LIN {X 0,Y 412.158,Z 270.316,A -85,B 0,C 180,E1 -10502.038,E2 -10502.038} C_VEL
LIN {X 0,Y 411.576,Z 278.2,A -85,B 0,C 180,E1 -10505.303,E2 -10505.303} C_VEL
LIN {X 0,Y 411.175,Z 285.935,A -85,B 0,C 180,E1 -10508.441,E2 -10508.441} C_VEL
LIN {X 0,Y 410.796,Z 293.73,A -85,B 0,C 180,E1 -10511.55,E2 -10511.55} C_VEL
LIN {X 0,Y 410.71,Z 295.781,A -85,B 0,C 180,E1 -10512.362,E2 -10512.362} C_VEL
LIN {X 0,Y 413.099,Z 311.021,A -85,B 0,C 180,E1 -10512.959,E2 -10512.959} C_VEL
LIN {X 0,Y 414.896,Z 323.777,A -85,B 0,C 180,E1 -10513.647,E2 -10513.647} C_VEL
LIN {X 0,Y 414.256,Z 335.412,A -85,B 0,C 180,E1 -10514.377,E2 -10514.377} C_VEL
LIN {X 0,Y 413.495,Z 346.072,A -85,B 0,C 180,E1 -10515.231,E2 -10515.231} C_VEL
LIN {X 0,Y 412.718,Z 356.985,A -85,B 0,C 180,E1 -10516.335,E2 -10516.335} C_VEL
LIN {X 0,Y 412.142,Z 365.905,A -85,B 0,C 180,E1 -10517.444,E2 -10517.444} C_VEL
LIN {X 0,Y 411.367,Z 375.608,A -85,B 0,C 180,E1 -10518.92,E2 -10518.92} C_VEL
LIN {X 0,Y 410.824,Z 383.345,A -85,B 0,C 180,E1 -10520.4,E2 -10520.4} C_VEL
LIN {X 0,Y 410.352,Z 390.488,A -85,B 0,C 180,E1 -10522.126,E2 -10522.126} C_VEL
LIN {X 0,Y 410.176,Z 395.252,A -85,B 0,C 180,E1 -10523.607,E2 -10523.607} C_VEL
LIN {X 0,Y 410.095,Z 398.897,A -85,B 0,C 180,E1 -10525.086,E2 -10525.086} C_VEL
LIN {X 0,Y 409.954,Z 400.772,A -85,B 0,C 180,E1 -10526.069,E2 -10526.069} C_VEL
LIN {X 0,Y 410.007,Z 402.189,A -85,B 0,C 180,E1 -10527.054,E2 -10527.054} C_VEL
LIN {X 0,Y 409.988,Z 403.197,A -85,B 0,C 180,E1 -10528.037,E2 -10528.037} C_VEL
LIN {X 0,Y 409.958,Z 403.812,A -85,B 0,C 180,E1 -10529.019,E2 -10529.019} C_VEL
LIN {X 0,Y 409.967,Z 404.032,A -85,B 0,C 180,E1 -10530.001,E2 -10530.001} C_VEL
LIN {X 0,Y 409.959,Z 403.815,A -85,B 0,C 180,E1 -10530.984,E2 -10530.984} C_VEL
LIN {X 0,Y 409.989,Z 403.204,A -85,B 0,C 180,E1 -10531.966,E2 -10531.966} C_VEL
LIN {X 0,Y 410.007,Z 402.201,A -85,B 0,C 180,E1 -10532.949,E2 -10532.949} C_VEL
LIN {X 0,Y 409.955,Z 400.787,A -85,B 0,C 180,E1 -10533.933,E2 -10533.933} C_VEL
LIN {X 0,Y 410.108,Z 397.83,A -85,B 0,C 180,E1 -10535.41,E2 -10535.41} C_VEL
LIN {X 0,Y 410.199,Z 393.819,A -85,B 0,C 180,E1 -10536.89,E2 -10536.89} C_VEL
LIN {X 0,Y 410.552,Z 387.661,A -85,B 0,C 180,E1 -10538.616,E2 -10538.616} C_VEL
LIN {X 0,Y 410.995,Z 380.937,A -85,B 0,C 180,E1 -10540.096,E2 -10540.096} C_VEL
LIN {X 0,Y 411.603,Z 372.598,A -85,B 0,C 180,E1 -10541.575,E2 -10541.575} C_VEL
LIN {X 0,Y 412.222,Z 364.05,A -85,B 0,C 180,E1 -10542.807,E2 -10542.807} C_VEL
LIN {X 0,Y 412.945,Z 354.466,A -85,B 0,C 180,E1 -10543.934,E2 -10543.934} C_VEL
LIN {X 0,Y 413.699,Z 343.045,A -85,B 0,C 180,E1 -10545.016,E2 -10545.016} C_VEL
LIN {X 0,Y 414.479,Z 331.604,A -85,B 0,C 180,E1 -10545.869,E2 -10545.869} C_VEL
LIN {X 0,Y 414.807,Z 323.36,A -85,B 0,C 180,E1 -10546.359,E2 -10546.359} C_VEL
LIN {X 0,Y 412.936,Z 309.911,A -85,B 0,C 180,E1 -10547.061,E2 -10547.061} C_VEL
LIN {X 0,Y 410.806,Z 297.017,A -85,B 0,C 180,E1 -10547.536,E2 -10547.536} C_VEL
LIN {X 0,Y 410.688,Z 295.908,A -85,B 0,C 180,E1 -10547.565,E2 -10547.565} C_VEL
LIN {X 0,Y 411.053,Z 288.417,A -85,B 0,C 180,E1 -10550.519,E2 -10550.519} C_VEL
LIN {X 0,Y 411.401,Z 280.488,A -85,B 0,C 180,E1 -10553.67,E2 -10553.67} C_VEL
LIN {X 0,Y 411.91,Z 272.527,A -85,B 0,C 180,E1 -10556.883,E2 -10556.883} C_VEL
LIN {X 0,Y 412.427,Z 264.541,A -85,B 0,C 180,E1 -10560.18,E2 -10560.18} C_VEL
LIN {X 0,Y 412.928,Z 257.914,A -85,B 0,C 180,E1 -10563.001,E2 -10563.001} C_VEL
LIN {X 0,Y 413.391,Z 251.345,A -85,B 0,C 180,E1 -10565.913,E2 -10565.913} C_VEL
LIN {X 0,Y 413.002,Z 247.385,A -85,B 0,C 180,E1 -10567.78,E2 -10567.78} C_VEL
LIN {X 0,Y 411.812,Z 240.314,A -85,B 0,C 180,E1 -10571.331,E2 -10571.331} C_VEL
LIN {X 0,Y 411.213,Z 237.266,A -85,B 0,C 180,E1 -10572.958,E2 -10572.958} C_VEL
LIN {X 0,Y 411.175,Z 237.273,A -85,B 0,C 180,E1 -10575.882,E2 -10575.882} C_VEL
LIN {X 0,Y 411.17,Z 237.27,A -85,B 0,C 180,E1 -10578.772,E2 -10578.772} C_VEL
LIN {X 0,Y 411.198,Z 237.263,A -85,B 0,C 180,E1 -10582.027,E2 -10582.027} C_VEL
LIN {X 0,Y 411.199,Z 237.261,A -85,B 0,C 180,E1 -10585.666,E2 -10585.666} C_VEL
LIN {X 0,Y 411.194,Z 237.263,A -85,B 0,C 180,E1 -10589.153,E2 -10589.153} C_VEL
LIN {X 0,Y 411.215,Z 237.263,A -85,B 0,C 180,E1 -10592.519,E2 -10592.519} C_VEL
LIN {X 0,Y 411.225,Z 237.262,A -85,B 0,C 180,E1 -10595.785,E2 -10595.785} C_VEL
LIN {X 0,Y 411.204,Z 237.262,A -85,B 0,C 180,E1 -10598.966,E2 -10598.966} C_VEL
LIN {X 0,Y 411.237,Z 237.262,A -85,B 0,C 180,E1 -10602.084,E2 -10602.084} C_VEL
LIN {X 0,Y 411.236,Z 237.257,A -85,B 0,C 180,E1 -10605.147,E2 -10605.147} C_VEL
LIN {X 0,Y 411.28,Z 237.254,A -85,B 0,C 180,E1 -10608.167,E2 -10608.167} C_VEL
LIN {X 0,Y 411.446,Z 237.234,A -85,B 0,C 180,E1 -10612.192,E2 -10612.192} C_VEL
LIN {X 0,Y 411.473,Z 237.231,A -85,B 0,C 180,E1 -10614.118,E2 -10614.118} C_VEL
LIN {X 0,Y 411.518,Z 237.225,A -85,B 0,C 180,E1 -10618.043,E2 -10618.043} C_VEL
LIN {X 0,Y 411.644,Z 237.209,A -85,B 0,C 180,E1 -10620,E2 -10620} C_VEL
LIN {X 0,Y 411.452,Z 237.232,A -85,B 0,C 180,E1 -10622.937,E2 -10622.937} C_VEL
LIN {X 0,Y 411.393,Z 237.239,A -85,B 0,C 180,E1 -10626.868,E2 -10626.868} C_VEL
LIN {X 0,Y 411.292,Z 237.252,A -85,B 0,C 180,E1 -10629.839,E2 -10629.839} C_VEL
LIN {X 0,Y 411.314,Z 237.252,A -85,B 0,C 180,E1 -10633.104,E2 -10633.104} C_VEL
LIN {X 0,Y 411.266,Z 237.257,A -85,B 0,C 180,E1 -10636.889,E2 -10636.889} C_VEL
LIN {X 0,Y 411.239,Z 237.258,A -85,B 0,C 180,E1 -10639.987,E2 -10639.987} C_VEL
LIN {X 0,Y 411.194,Z 237.266,A -85,B 0,C 180,E1 -10643.148,E2 -10643.148} C_VEL
LIN {X 0,Y 411.171,Z 237.267,A -85,B 0,C 180,E1 -10646.386,E2 -10646.386} C_VEL
LIN {X 0,Y 411.204,Z 237.261,A -85,B 0,C 180,E1 -10649.713,E2 -10649.713} C_VEL
LIN {X 0,Y 411.214,Z 237.262,A -85,B 0,C 180,E1 -10653.155,E2 -10653.155} C_VEL
LIN {X 0,Y 411.199,Z 237.266,A -85,B 0,C 180,E1 -10656.552,E2 -10656.552} C_VEL
LIN {X 0,Y 411.214,Z 237.262,A -85,B 0,C 180,E1 -10659.726,E2 -10659.726} C_VEL
LIN {X 0,Y 411.178,Z 237.265,A -85,B 0,C 180,E1 -10663.133,E2 -10663.133} C_VEL
LIN {X 0,Y 411.17,Z 237.268,A -85,B 0,C 180,E1 -10665.881,E2 -10665.881} C_VEL
LIN {X 0,Y 411.164,Z 237.267,A -85,B 0,C 180,E1 -10669.492,E2 -10669.492} C_VEL
LIN {X 0,Y 411.192,Z 237.267,A -85,B 0,C 180,E1 -10672.024,E2 -10672.024} C_VEL
LIN {X 0,Y 411.21,Z 237.262,A -85,B 0,C 180,E1 -10675.122,E2 -10675.122} C_VEL
LIN {X 0,Y 411.107,Z 237.277,A -85,B 0,C 180,E1 -10677.996,E2 -10677.996} C_VEL
LIN {X 0,Y 410.789,Z 237.318,A -85,B 0,C 180,E1 -10681.376,E2 -10681.376} C_VEL
LIN {X 0,Y 410.632,Z 237.497,A -85,B 0,C 180,E1 -10682.872,E2 -10682.872} C_VEL
LIN {X 0,Y 410.568,Z 240.288,A -85,B 0,C 180,E1 -10685.742,E2 -10685.742} C_VEL
LIN {X 0,Y 410.475,Z 243.402,A -85,B 0,C 180,E1 -10688.926,E2 -10688.926} C_VEL
LIN {X 0,Y 410.409,Z 246.589,A -85,B 0,C 180,E1 -10692.045,E2 -10692.045} C_VEL
LIN {X 0,Y 410.381,Z 249.825,A -85,B 0,C 180,E1 -10695.113,E2 -10695.113} C_VEL
LIN {X 0,Y 410.411,Z 251.602,A -85,B 0,C 180,E1 -10696.745,E2 -10696.745} C_VEL
LIN {X 0,Y 413.741,Z 265.221,A -85,B 0,C 180,E1 -10697.347,E2 -10697.347} C_VEL
LIN {X 0,Y 415.318,Z 272.966,A -85,B 0,C 180,E1 -10697.776,E2 -10697.776} C_VEL
LIN {X 0,Y 414.783,Z 285.252,A -85,B 0,C 180,E1 -10698.515,E2 -10698.515} C_VEL
LIN {X 0,Y 414.047,Z 297.573,A -85,B 0,C 180,E1 -10699.485,E2 -10699.485} C_VEL
LIN {X 0,Y 413.416,Z 307.511,A -85,B 0,C 180,E1 -10700.482,E2 -10700.482} C_VEL
LIN {X 0,Y 412.804,Z 317.143,A -85,B 0,C 180,E1 -10701.678,E2 -10701.678} C_VEL
LIN {X 0,Y 412.051,Z 326.69,A -85,B 0,C 180,E1 -10703.142,E2 -10703.142} C_VEL
LIN {X 0,Y 411.438,Z 334.306,A -85,B 0,C 180,E1 -10704.608,E2 -10704.608} C_VEL
LIN {X 0,Y 410.884,Z 340.421,A -85,B 0,C 180,E1 -10706.075,E2 -10706.075} C_VEL
LIN {X 0,Y 410.502,Z 345.28,A -85,B 0,C 180,E1 -10707.545,E2 -10707.545} C_VEL
LIN {X 0,Y 410.231,Z 349.036,A -85,B 0,C 180,E1 -10709.017,E2 -10709.017} C_VEL
LIN {X 0,Y 410.163,Z 350.969,A -85,B 0,C 180,E1 -10709.999,E2 -10709.999} C_VEL
LIN {X 0,Y 410.148,Z 352.495,A -85,B 0,C 180,E1 -10710.98,E2 -10710.98} C_VEL
LIN {X 0,Y 410.143,Z 353.592,A -85,B 0,C 180,E1 -10711.963,E2 -10711.963} C_VEL
LIN {X 0,Y 410.195,Z 354.28,A -85,B 0,C 180,E1 -10712.945,E2 -10712.945} C_VEL
LIN {X 0,Y 410.11,Z 354.543,A -85,B 0,C 180,E1 -10714.914,E2 -10714.914} C_VEL
LIN {X 0,Y 410.212,Z 353.644,A -85,B 0,C 180,E1 -10716.435,E2 -10716.435} C_VEL
LIN {X 0,Y 410.296,Z 351.92,A -85,B 0,C 180,E1 -10717.875,E2 -10717.875} C_VEL
LIN {X 0,Y 410.485,Z 348.979,A -85,B 0,C 180,E1 -10719.466,E2 -10719.466} C_VEL
LIN {X 0,Y 409.963,Z 347.209,A -85,B 0,C 180,E1 -10720.249,E2 -10720.249} C_VEL
LIN {X 0,Y 407.393,Z 343.929,A -85,B 0,C 180,E1 -10721.513,E2 -10721.513} C_VEL
LIN {X 0,Y 404.911,Z 340.075,A -85,B 0,C 180,E1 -10722.754,E2 -10722.754} C_VEL
LIN {X 0,Y 404.534,Z 337.241,A -85,B 0,C 180,E1 -10723.49,E2 -10723.49} C_VEL
LIN {X 0,Y 405.238,Z 329.743,A -85,B 0,C 180,E1 -10725.077,E2 -10725.077} C_VEL
LIN {X 0,Y 406.067,Z 320.767,A -85,B 0,C 180,E1 -10726.592,E2 -10726.592} C_VEL
LIN {X 0,Y 406.922,Z 311.461,A -85,B 0,C 180,E1 -10727.851,E2 -10727.851} C_VEL
LIN {X 0,Y 407.693,Z 301.065,A -85,B 0,C 180,E1 -10728.987,E2 -10728.987} C_VEL
LIN {X 0,Y 408.603,Z 289.481,A -85,B 0,C 180,E1 -10729.988,E2 -10729.988} C_VEL
LIN {X 0,Y 409.132,Z 277.866,A -85,B 0,C 180,E1 -10730.774,E2 -10730.774} C_VEL
LIN {X 0,Y 409.283,Z 275.137,A -85,B 0,C 180,E1 -10730.924,E2 -10730.924} C_VEL
LIN {X 0,Y 406.594,Z 263.548,A -85,B 0,C 180,E1 -10731.625,E2 -10731.625} C_VEL
LIN {X 0,Y 403.358,Z 252.181,A -85,B 0,C 180,E1 -10732.198,E2 -10732.198} C_VEL
LIN {X 0,Y 403.446,Z 248.467,A -85,B 0,C 180,E1 -10735.815,E2 -10735.815} C_VEL
LIN {X 0,Y 403.577,Z 244.876,A -85,B 0,C 180,E1 -10739.458,E2 -10739.458} C_VEL
LIN {X 0,Y 403.601,Z 241.861,A -85,B 0,C 180,E1 -10742.669,E2 -10742.669} C_VEL
LIN {X 0,Y 403.723,Z 239.598,A -85,B 0,C 180,E1 -10745.097,E2 -10745.097} C_VEL
LIN {X 0,Y 403.816,Z 238.188,A -85,B 0,C 180,E1 -10746.814,E2 -10746.814} C_VEL
LIN {X 0,Y 404.085,Z 238.149,A -85,B 0,C 180,E1 -10750.069,E2 -10750.069} C_VEL
LIN {X 0,Y 404.145,Z 238.144,A -85,B 0,C 180,E1 -10753.082,E2 -10753.082} C_VEL
LIN {X 0,Y 404.14,Z 238.146,A -85,B 0,C 180,E1 -10755.925,E2 -10755.925} C_VEL
LIN {X 0,Y 404.107,Z 238.148,A -85,B 0,C 180,E1 -10758.633,E2 -10758.633} C_VEL
LIN {X 0,Y 404.145,Z 238.142,A -85,B 0,C 180,E1 -10761.491,E2 -10761.491} C_VEL
LIN {X 0,Y 404.177,Z 238.138,A -85,B 0,C 180,E1 -10764.983,E2 -10764.983} C_VEL
LIN {X 0,Y 404.132,Z 238.143,A -85,B 0,C 180,E1 -10768.553,E2 -10768.553} C_VEL
LIN {X 0,Y 404.186,Z 238.137,A -85,B 0,C 180,E1 -10771.999,E2 -10771.999} C_VEL
LIN {X 0,Y 404.167,Z 238.14,A -85,B 0,C 180,E1 -10775.333,E2 -10775.333} C_VEL
LIN {X 0,Y 404.128,Z 238.145,A -85,B 0,C 180,E1 -10778.58,E2 -10778.58} C_VEL
LIN {X 0,Y 404.199,Z 238.135,A -85,B 0,C 180,E1 -10781.761,E2 -10781.761} C_VEL
LIN {X 0,Y 404.195,Z 238.136,A -85,B 0,C 180,E1 -10784.881,E2 -10784.881} C_VEL
LIN {X 0,Y 404.244,Z 238.129,A -85,B 0,C 180,E1 -10787.958,E2 -10787.958} C_VEL
LIN {X 0,Y 404.422,Z 238.111,A -85,B 0,C 180,E1 -10792.099,E2 -10792.099} C_VEL
LIN {X 0,Y 404.429,Z 238.111,A -85,B 0,C 180,E1 -10794.015,E2 -10794.015} C_VEL
LIN {X 0,Y 404.472,Z 238.101,A -85,B 0,C 180,E1 -10798.008,E2 -10798.008} C_VEL
LIN {X 0,Y 404.596,Z 238.087,A -85,B 0,C 180,E1 -10800,E2 -10800} C_VEL
LIN {X 0,Y 404.413,Z 238.109,A -85,B 0,C 180,E1 -10802.988,E2 -10802.988} C_VEL
LIN {X 0,Y 404.428,Z 238.107,A -85,B 0,C 180,E1 -10805.985,E2 -10805.985} C_VEL
LIN {X 0,Y 404.411,Z 238.109,A -85,B 0,C 180,E1 -10807.991,E2 -10807.991} C_VEL
LIN {X 0,Y 404.244,Z 238.133,A -85,B 0,C 180,E1 -10812.042,E2 -10812.042} C_VEL
LIN {X 0,Y 404.194,Z 238.136,A -85,B 0,C 180,E1 -10815.118,E2 -10815.118} C_VEL
LIN {X 0,Y 404.199,Z 238.136,A -85,B 0,C 180,E1 -10818.239,E2 -10818.239} C_VEL
LIN {X 0,Y 404.127,Z 238.145,A -85,B 0,C 180,E1 -10821.42,E2 -10821.42} C_VEL
LIN {X 0,Y 404.166,Z 238.14,A -85,B 0,C 180,E1 -10824.666,E2 -10824.666} C_VEL
LIN {X 0,Y 404.188,Z 238.138,A -85,B 0,C 180,E1 -10828,E2 -10828} C_VEL
LIN {X 0,Y 404.136,Z 238.146,A -85,B 0,C 180,E1 -10831.56,E2 -10831.56} C_VEL
LIN {X 0,Y 404.175,Z 238.139,A -85,B 0,C 180,E1 -10835.017,E2 -10835.017} C_VEL
LIN {X 0,Y 404.145,Z 238.144,A -85,B 0,C 180,E1 -10838.758,E2 -10838.758} C_VEL
LIN {X 0,Y 404.11,Z 238.149,A -85,B 0,C 180,E1 -10841.6,E2 -10841.6} C_VEL
LIN {X 0,Y 404.137,Z 238.146,A -85,B 0,C 180,E1 -10844.523,E2 -10844.523} C_VEL
LIN {X 0,Y 404.152,Z 238.286,A -85,B 0,C 180,E1 -10845.839,E2 -10845.839} C_VEL
LIN {X 0,Y 405.143,Z 243.346,A -85,B 0,C 180,E1 -10848.765,E2 -10848.765} C_VEL
LIN {X 0,Y 406.197,Z 249.585,A -85,B 0,C 180,E1 -10852.108,E2 -10852.108} C_VEL
LIN {X 0,Y 406.557,Z 253.389,A -85,B 0,C 180,E1 -10854.005,E2 -10854.005} C_VEL
LIN {X 0,Y 406.046,Z 259.761,A -85,B 0,C 180,E1 -10856.963,E2 -10856.963} C_VEL
LIN {X 0,Y 405.374,Z 266.817,A -85,B 0,C 180,E1 -10860.095,E2 -10860.095} C_VEL
LIN {X 0,Y 404.903,Z 273.956,A -85,B 0,C 180,E1 -10863.175,E2 -10863.175} C_VEL
LIN {X 0,Y 404.259,Z 283.395,A -85,B 0,C 180,E1 -10867.132,E2 -10867.132} C_VEL
LIN {X 0,Y 403.903,Z 290.359,A -85,B 0,C 180,E1 -10869.987,E2 -10869.987} C_VEL
LIN {X 0,Y 403.661,Z 295.493,A -85,B 0,C 180,E1 -10872.05,E2 -10872.05} C_VEL
LIN {X 0,Y 405.902,Z 308.96,A -85,B 0,C 180,E1 -10872.562,E2 -10872.562} C_VEL
LIN {X 0,Y 407.69,Z 321.978,A -85,B 0,C 180,E1 -10873.257,E2 -10873.257} C_VEL
LIN {X 0,Y 408.009,Z 326.19,A -85,B 0,C 180,E1 -10873.515,E2 -10873.515} C_VEL
LIN {X 0,Y 407.144,Z 338.416,A -85,B 0,C 180,E1 -10874.354,E2 -10874.354} C_VEL
LIN {X 0,Y 406.287,Z 350.067,A -85,B 0,C 180,E1 -10875.386,E2 -10875.386} C_VEL
LIN {X 0,Y 405.557,Z 359.842,A -85,B 0,C 180,E1 -10876.472,E2 -10876.472} C_VEL
LIN {X 0,Y 404.878,Z 369.022,A -85,B 0,C 180,E1 -10877.725,E2 -10877.725} C_VEL
LIN {X 0,Y 404.114,Z 377.979,A -85,B 0,C 180,E1 -10879.226,E2 -10879.226} C_VEL
LIN {X 0,Y 403.611,Z 385.201,A -85,B 0,C 180,E1 -10880.733,E2 -10880.733} C_VEL
LIN {X 0,Y 403.299,Z 390.084,A -85,B 0,C 180,E1 -10881.988,E2 -10881.988} C_VEL
LIN {X 0,Y 403.068,Z 395.288,A -85,B 0,C 180,E1 -10883.652,E2 -10883.652} C_VEL
LIN {X 0,Y 403.007,Z 398.478,A -85,B 0,C 180,E1 -10884.999,E2 -10884.999} C_VEL
LIN {X 0,Y 402.877,Z 400.351,A -85,B 0,C 180,E1 -10886,E2 -10886} C_VEL
LIN {X 0,Y 402.908,Z 401.764,A -85,B 0,C 180,E1 -10887.002,E2 -10887.002} C_VEL
LIN {X 0,Y 402.921,Z 402.773,A -85,B 0,C 180,E1 -10888.002,E2 -10888.002} C_VEL
LIN {X 0,Y 402.884,Z 403.387,A -85,B 0,C 180,E1 -10889.002,E2 -10889.002} C_VEL
LIN {X 0,Y 402.89,Z 403.606,A -85,B 0,C 180,E1 -10890.001,E2 -10890.001} C_VEL
LIN {X 0,Y 402.921,Z 402.776,A -85,B 0,C 180,E1 -10892.001,E2 -10892.001} C_VEL
LIN {X 0,Y 402.909,Z 401.769,A -85,B 0,C 180,E1 -10893.001,E2 -10893.001} C_VEL
LIN {X 0,Y 402.877,Z 400.354,A -85,B 0,C 180,E1 -10894.003,E2 -10894.003} C_VEL
LIN {X 0,Y 403.007,Z 397.391,A -85,B 0,C 180,E1 -10895.505,E2 -10895.505} C_VEL
LIN {X 0,Y 403.118,Z 393.373,A -85,B 0,C 180,E1 -10897.011,E2 -10897.011} C_VEL
LIN {X 0,Y 403.518,Z 387.204,A -85,B 0,C 180,E1 -10898.767,E2 -10898.767} C_VEL
LIN {X 0,Y 403.967,Z 380.466,A -85,B 0,C 180,E1 -10900.274,E2 -10900.274} C_VEL
LIN {X 0,Y 404.61,Z 372.111,A -85,B 0,C 180,E1 -10901.778,E2 -10901.778} C_VEL
LIN {X 0,Y 405.238,Z 363.536,A -85,B 0,C 180,E1 -10903.031,E2 -10903.031} C_VEL
LIN {X 0,Y 406.022,Z 353.452,A -85,B 0,C 180,E1 -10904.227,E2 -10904.227} C_VEL
LIN {X 0,Y 406.791,Z 342.474,A -85,B 0,C 180,E1 -10905.277,E2 -10905.277} C_VEL
LIN {X 0,Y 407.637,Z 331.106,A -85,B 0,C 180,E1 -10906.134,E2 -10906.134} C_VEL
LIN {X 0,Y 407.919,Z 324.481,A -85,B 0,C 180,E1 -10906.542,E2 -10906.542} C_VEL
LIN {X 0,Y 406.056,Z 310.699,A -85,B 0,C 180,E1 -10907.292,E2 -10907.292} C_VEL
LIN {X 0,Y 403.915,Z 297.479,A -85,B 0,C 180,E1 -10907.808,E2 -10907.808} C_VEL
LIN {X 0,Y 403.625,Z 295.48,A -85,B 0,C 180,E1 -10907.873,E2 -10907.873} C_VEL
LIN {X 0,Y 404.072,Z 286.681,A -85,B 0,C 180,E1 -10911.425,E2 -10911.425} C_VEL
LIN {X 0,Y 404.628,Z 276.913,A -85,B 0,C 180,E1 -10915.419,E2 -10915.419} C_VEL
LIN {X 0,Y 405.137,Z 269.504,A -85,B 0,C 180,E1 -10918.494,E2 -10918.494} C_VEL
LIN {X 0,Y 405.753,Z 261.477,A -85,B 0,C 180,E1 -10921.927,E2 -10921.927} C_VEL
LIN {X 0,Y 406.26,Z 254.965,A -85,B 0,C 180,E1 -10924.813,E2 -10924.813} C_VEL
LIN {X 0,Y 406.334,Z 251.056,A -85,B 0,C 180,E1 -10926.629,E2 -10926.629} C_VEL
LIN {X 0,Y 405.527,Z 245.689,A -85,B 0,C 180,E1 -10929.29,E2 -10929.29} C_VEL
LIN {X 0,Y 404.417,Z 239.27,A -85,B 0,C 180,E1 -10932.669,E2 -10932.669} C_VEL
LIN {X 0,Y 404.159,Z 238.146,A -85,B 0,C 180,E1 -10933.338,E2 -10933.338} C_VEL
LIN {X 0,Y 404.16,Z 238.143,A -85,B 0,C 180,E1 -10936.917,E2 -10936.917} C_VEL
LIN {X 0,Y 404.176,Z 238.14,A -85,B 0,C 180,E1 -10939.956,E2 -10939.956} C_VEL
LIN {X 0,Y 404.142,Z 238.142,A -85,B 0,C 180,E1 -10943.126,E2 -10943.126} C_VEL
LIN {X 0,Y 404.144,Z 238.143,A -85,B 0,C 180,E1 -10946.188,E2 -10946.188} C_VEL
LIN {X 0,Y 404.15,Z 238.14,A -85,B 0,C 180,E1 -10949.715,E2 -10949.715} C_VEL
LIN {X 0,Y 404.158,Z 238.14,A -85,B 0,C 180,E1 -10953.12,E2 -10953.12} C_VEL
LIN {X 0,Y 404.173,Z 238.141,A -85,B 0,C 180,E1 -10956.426,E2 -10956.426} C_VEL
LIN {X 0,Y 404.199,Z 238.137,A -85,B 0,C 180,E1 -10959.875,E2 -10959.875} C_VEL
LIN {X 0,Y 404.181,Z 238.136,A -85,B 0,C 180,E1 -10963.013,E2 -10963.013} C_VEL
LIN {X 0,Y 404.291,Z 238.122,A -85,B 0,C 180,E1 -10966.939,E2 -10966.939} C_VEL
LIN {X 0,Y 404.252,Z 238.131,A -85,B 0,C 180,E1 -10969.988,E2 -10969.988} C_VEL
LIN {X 0,Y 404.393,Z 238.111,A -85,B 0,C 180,E1 -10973.013,E2 -10973.013} C_VEL
LIN {X 0,Y 404.285,Z 238.124,A -85,B 0,C 180,E1 -10975.014,E2 -10975.014} C_VEL
LIN {X 0,Y 404.487,Z 238.101,A -85,B 0,C 180,E1 -10978.009,E2 -10978.009} C_VEL
LIN {X 0,Y 404.613,Z 238.085,A -85,B 0,C 180,E1 -10980,E2 -10980} C_VEL
LIN {X 0,Y 404.41,Z 238.11,A -85,B 0,C 180,E1 -10982.989,E2 -10982.989} C_VEL
LIN {X 0,Y 404.344,Z 238.118,A -85,B 0,C 180,E1 -10986.989,E2 -10986.989} C_VEL
LIN {X 0,Y 404.258,Z 238.127,A -85,B 0,C 180,E1 -10990.012,E2 -10990.012} C_VEL
LIN {X 0,Y 404.275,Z 238.128,A -85,B 0,C 180,E1 -10993.211,E2 -10993.211} C_VEL
LIN {X 0,Y 404.224,Z 238.135,A -85,B 0,C 180,E1 -10997.007,E2 -10997.007} C_VEL
LIN {X 0,Y 404.172,Z 238.139,A -85,B 0,C 180,E1 -11000.351,E2 -11000.351} C_VEL
LIN {X 0,Y 404.155,Z 238.14,A -85,B 0,C 180,E1 -11003.576,E2 -11003.576} C_VEL
LIN {X 0,Y 404.105,Z 238.149,A -85,B 0,C 180,E1 -11006.884,E2 -11006.884} C_VEL
LIN {X 0,Y 404.151,Z 238.143,A -85,B 0,C 180,E1 -11010.285,E2 -11010.285} C_VEL
LIN {X 0,Y 404.152,Z 238.141,A -85,B 0,C 180,E1 -11013.812,E2 -11013.812} C_VEL
LIN {X 0,Y 404.142,Z 238.144,A -85,B 0,C 180,E1 -11016.874,E2 -11016.874} C_VEL
LIN {X 0,Y 404.155,Z 238.143,A -85,B 0,C 180,E1 -11020.08,E2 -11020.08} C_VEL
LIN {X 0,Y 404.157,Z 238.139,A -85,B 0,C 180,E1 -11023.083,E2 -11023.083} C_VEL
LIN {X 0,Y 404.127,Z 238.146,A -85,B 0,C 180,E1 -11025.921,E2 -11025.921} C_VEL
LIN {X 0,Y 404.107,Z 238.146,A -85,B 0,C 180,E1 -11028.632,E2 -11028.632} C_VEL
LIN {X 0,Y 404.146,Z 238.142,A -85,B 0,C 180,E1 -11031.494,E2 -11031.494} C_VEL
LIN {X 0,Y 404.181,Z 238.137,A -85,B 0,C 180,E1 -11034.982,E2 -11034.982} C_VEL
LIN {X 0,Y 404.106,Z 238.148,A -85,B 0,C 180,E1 -11037.374,E2 -11037.374} C_VEL
LIN {X 0,Y 403.861,Z 238.177,A -85,B 0,C 180,E1 -11040.471,E2 -11040.471} C_VEL
LIN {X 0,Y 403.581,Z 238.217,A -85,B 0,C 180,E1 -11042.639,E2 -11042.639} C_VEL
LIN {X 0,Y 403.551,Z 240.636,A -85,B 0,C 180,E1 -11045.292,E2 -11045.292} C_VEL
LIN {X 0,Y 403.409,Z 243.794,A -85,B 0,C 180,E1 -11048.539,E2 -11048.539} C_VEL
LIN {X 0,Y 403.349,Z 247.016,A -85,B 0,C 180,E1 -11051.72,E2 -11051.72} C_VEL
LIN {X 0,Y 403.368,Z 249.156,A -85,B 0,C 180,E1 -11053.812,E2 -11053.812} C_VEL
LIN {X 0,Y 403.343,Z 252.005,A -85,B 0,C 180,E1 -11056.457,E2 -11056.457} C_VEL
LIN {X 0,Y 406.664,Z 265.573,A -85,B 0,C 180,E1 -11057.069,E2 -11057.069} C_VEL
LIN {X 0,Y 408.436,Z 274.588,A -85,B 0,C 180,E1 -11057.586,E2 -11057.586} C_VEL
LIN {X 0,Y 407.891,Z 286.345,A -85,B 0,C 180,E1 -11058.318,E2 -11058.318} C_VEL
LIN {X 0,Y 407.222,Z 297.129,A -85,B 0,C 180,E1 -11059.181,E2 -11059.181} C_VEL
LIN {X 0,Y 406.486,Z 308.339,A -85,B 0,C 180,E1 -11060.318,E2 -11060.318} C_VEL
LIN {X 0,Y 405.838,Z 317.906,A -85,B 0,C 180,E1 -11061.534,E2 -11061.534} C_VEL
LIN {X 0,Y 405.055,Z 327.394,A -85,B 0,C 180,E1 -11063.022,E2 -11063.022} C_VEL
LIN {X 0,Y 404.413,Z 334.944,A -85,B 0,C 180,E1 -11064.514,E2 -11064.514} C_VEL
LIN {X 0,Y 403.825,Z 341.021,A -85,B 0,C 180,E1 -11066.007,E2 -11066.007} C_VEL
LIN {X 0,Y 403.445,Z 345.842,A -85,B 0,C 180,E1 -11067.503,E2 -11067.503} C_VEL
LIN {X 0,Y 403.175,Z 349.562,A -85,B 0,C 180,E1 -11069,E2 -11069} C_VEL
LIN {X 0,Y 403.106,Z 351.479,A -85,B 0,C 180,E1 -11069.999,E2 -11069.999} C_VEL
LIN {X 0,Y 403.063,Z 352.989,A -85,B 0,C 180,E1 -11070.998,E2 -11070.998} C_VEL
LIN {X 0,Y 403.126,Z 354.729,A -85,B 0,C 180,E1 -11072.997,E2 -11072.997} C_VEL
LIN {X 0,Y 403.045,Z 354.961,A -85,B 0,C 180,E1 -11075,E2 -11075} C_VEL
LIN {X 0,Y 403.143,Z 354.118,A -85,B 0,C 180,E1 -11076.44,E2 -11076.44} C_VEL
LIN {X 0,Y 403.234,Z 352.279,A -85,B 0,C 180,E1 -11078.013,E2 -11078.013} C_VEL
LIN {X 0,Y 403.435,Z 349.545,A -85,B 0,C 180,E1 -11079.524,E2 -11079.524} C_VEL
LIN {X 0,Y 403.7,Z 345.791,A -85,B 0,C 180,E1 -11081.039,E2 -11081.039} C_VEL
LIN {X 0,Y 404.192,Z 340.9,A -85,B 0,C 180,E1 -11082.552,E2 -11082.552} C_VEL
LIN {X 0,Y 404.534,Z 337.241,A -85,B 0,C 180,E1 -11083.49,E2 -11083.49} C_VEL
LIN {X 0,Y 404.192,Z 334.23,A -85,B 0,C 180,E1 -11084.209,E2 -11084.209} C_VEL
LIN {X 0,Y 401.912,Z 329.06,A -85,B 0,C 180,E1 -11085.369,E2 -11085.369} C_VEL
LIN {X 0,Y 399.656,Z 323.297,A -85,B 0,C 180,E1 -11086.478,E2 -11086.478} C_VEL
LIN {X 0,Y 399.352,Z 319.357,A -85,B 0,C 180,E1 -11087.108,E2 -11087.108} C_VEL
LIN {X 0,Y 400.243,Z 309.342,A -85,B 0,C 180,E1 -11088.424,E2 -11088.424} C_VEL
LIN {X 0,Y 401.077,Z 299.707,A -85,B 0,C 180,E1 -11089.445,E2 -11089.445} C_VEL
LIN {X 0,Y 401.879,Z 289.302,A -85,B 0,C 180,E1 -11090.337,E2 -11090.337} C_VEL
LIN {X 0,Y 402.433,Z 277.434,A -85,B 0,C 180,E1 -11091.136,E2 -11091.136} C_VEL
LIN {X 0,Y 402.289,Z 274.943,A -85,B 0,C 180,E1 -11091.29,E2 -11091.29} C_VEL
LIN {X 0,Y 399.109,Z 262.358,A -85,B 0,C 180,E1 -11092.063,E2 -11092.063} C_VEL
LIN {X 0,Y 396.284,Z 252.618,A -85,B 0,C 180,E1 -11092.55,E2 -11092.55} C_VEL
LIN {X 0,Y 396.391,Z 249.817,A -85,B 0,C 180,E1 -11095.279,E2 -11095.279} C_VEL
LIN {X 0,Y 396.484,Z 246.574,A -85,B 0,C 180,E1 -11098.592,E2 -11098.592} C_VEL
LIN {X 0,Y 396.534,Z 243.232,A -85,B 0,C 180,E1 -11102.119,E2 -11102.119} C_VEL
LIN {X 0,Y 396.676,Z 240.227,A -85,B 0,C 180,E1 -11105.413,E2 -11105.413} C_VEL
LIN {X 0,Y 396.819,Z 239.059,A -85,B 0,C 180,E1 -11107.156,E2 -11107.156} C_VEL
LIN {X 0,Y 397.033,Z 239.028,A -85,B 0,C 180,E1 -11110.433,E2 -11110.433} C_VEL
LIN {X 0,Y 397.094,Z 239.021,A -85,B 0,C 180,E1 -11113.647,E2 -11113.647} C_VEL
LIN {X 0,Y 397.094,Z 239.022,A -85,B 0,C 180,E1 -11116.52,E2 -11116.52} C_VEL
LIN {X 0,Y 397.105,Z 239.02,A -85,B 0,C 180,E1 -11120.421,E2 -11120.421} C_VEL
LIN {X 0,Y 397.101,Z 239.022,A -85,B 0,C 180,E1 -11124.264,E2 -11124.264} C_VEL
LIN {X 0,Y 397.105,Z 239.018,A -85,B 0,C 180,E1 -11126.726,E2 -11126.726} C_VEL
LIN {X 0,Y 397.115,Z 239.017,A -85,B 0,C 180,E1 -11130.295,E2 -11130.295} C_VEL
LIN {X 0,Y 397.185,Z 239.008,A -85,B 0,C 180,E1 -11132.609,E2 -11132.609} C_VEL
LIN {X 0,Y 397.123,Z 239.02,A -85,B 0,C 180,E1 -11135.981,E2 -11135.981} C_VEL
LIN {X 0,Y 397.128,Z 239.016,A -85,B 0,C 180,E1 -11139.704,E2 -11139.704} C_VEL
LIN {X 0,Y 397.171,Z 239.011,A -85,B 0,C 180,E1 -11142.844,E2 -11142.844} C_VEL
LIN {X 0,Y 397.217,Z 239.004,A -85,B 0,C 180,E1 -11146.702,E2 -11146.702} C_VEL
LIN {X 0,Y 397.205,Z 239.007,A -85,B 0,C 180,E1 -11149.808,E2 -11149.808} C_VEL
LIN {X 0,Y 397.354,Z 238.987,A -85,B 0,C 180,E1 -11152.888,E2 -11152.888} C_VEL
LIN {X 0,Y 397.253,Z 239.001,A -85,B 0,C 180,E1 -11154.925,E2 -11154.925} C_VEL
LIN {X 0,Y 397.441,Z 238.976,A -85,B 0,C 180,E1 -11157.973,E2 -11157.973} C_VEL
LIN {X 0,Y 397.565,Z 238.962,A -85,B 0,C 180,E1 -11160,E2 -11160} C_VEL
LIN {X 0,Y 397.372,Z 238.986,A -85,B 0,C 180,E1 -11163.041,E2 -11163.041} C_VEL
LIN {X 0,Y 397.377,Z 238.985,A -85,B 0,C 180,E1 -11166.091,E2 -11166.091} C_VEL
LIN {X 0,Y 397.365,Z 238.987,A -85,B 0,C 180,E1 -11168.134,E2 -11168.134} C_VEL
LIN {X 0,Y 397.207,Z 239.007,A -85,B 0,C 180,E1 -11172.258,E2 -11172.258} C_VEL
LIN {X 0,Y 397.167,Z 239.009,A -85,B 0,C 180,E1 -11175.392,E2 -11175.392} C_VEL
LIN {X 0,Y 397.151,Z 239.013,A -85,B 0,C 180,E1 -11178.574,E2 -11178.574} C_VEL
LIN {X 0,Y 397.086,Z 239.024,A -85,B 0,C 180,E1 -11181.819,E2 -11181.819} C_VEL
LIN {X 0,Y 397.146,Z 239.018,A -85,B 0,C 180,E1 -11185.132,E2 -11185.132} C_VEL
LIN {X 0,Y 397.153,Z 239.013,A -85,B 0,C 180,E1 -11187.777,E2 -11187.777} C_VEL
LIN {X 0,Y 397.076,Z 239.023,A -85,B 0,C 180,E1 -11190.883,E2 -11190.883} C_VEL
LIN {X 0,Y 397.116,Z 239.019,A -85,B 0,C 180,E1 -11194.494,E2 -11194.494} C_VEL
LIN {X 0,Y 397.093,Z 239.023,A -85,B 0,C 180,E1 -11198.276,E2 -11198.276} C_VEL
LIN {X 0,Y 397.078,Z 239.023,A -85,B 0,C 180,E1 -11200.91,E2 -11200.91} C_VEL
LIN {X 0,Y 397.092,Z 239.023,A -85,B 0,C 180,E1 -11203.65,E2 -11203.65} C_VEL
LIN {X 0,Y 397.115,Z 239.184,A -85,B 0,C 180,E1 -11205.425,E2 -11205.425} C_VEL
LIN {X 0,Y 398.154,Z 244.487,A -85,B 0,C 180,E1 -11208.579,E2 -11208.579} C_VEL
LIN {X 0,Y 399.025,Z 249.632,A -85,B 0,C 180,E1 -11211.398,E2 -11211.398} C_VEL
LIN {X 0,Y 399.552,Z 253.233,A -85,B 0,C 180,E1 -11213.272,E2 -11213.272} C_VEL
LIN {X 0,Y 399.293,Z 258.51,A -85,B 0,C 180,E1 -11215.818,E2 -11215.818} C_VEL
LIN {X 0,Y 398.518,Z 265.978,A -85,B 0,C 180,E1 -11219.243,E2 -11219.243} C_VEL
LIN {X 0,Y 397.943,Z 273.702,A -85,B 0,C 180,E1 -11222.668,E2 -11222.668} C_VEL
LIN {X 0,Y 397.372,Z 281.442,A -85,B 0,C 180,E1 -11225.999,E2 -11225.999} C_VEL
LIN {X 0,Y 396.943,Z 289.174,A -85,B 0,C 180,E1 -11229.263,E2 -11229.263} C_VEL
LIN {X 0,Y 396.603,Z 294.94,A -85,B 0,C 180,E1 -11231.669,E2 -11231.669} C_VEL
LIN {X 0,Y 399.153,Z 310.285,A -85,B 0,C 180,E1 -11232.312,E2 -11232.312} C_VEL
LIN {X 0,Y 400.892,Z 323.458,A -85,B 0,C 180,E1 -11233.057,E2 -11233.057} C_VEL
LIN {X 0,Y 401.085,Z 328.171,A -85,B 0,C 180,E1 -11233.363,E2 -11233.363} C_VEL
LIN {X 0,Y 400.198,Z 339.785,A -85,B 0,C 180,E1 -11234.206,E2 -11234.206} C_VEL
LIN {X 0,Y 399.256,Z 351.119,A -85,B 0,C 180,E1 -11235.266,E2 -11235.266} C_VEL
LIN {X 0,Y 398.43,Z 361.672,A -85,B 0,C 180,E1 -11236.509,E2 -11236.509} C_VEL
LIN {X 0,Y 397.754,Z 370.327,A -85,B 0,C 180,E1 -11237.76,E2 -11237.76} C_VEL
LIN {X 0,Y 397.015,Z 378.942,A -85,B 0,C 180,E1 -11239.29,E2 -11239.29} C_VEL
LIN {X 0,Y 396.497,Z 385.854,A -85,B 0,C 180,E1 -11240.822,E2 -11240.822} C_VEL
LIN {X 0,Y 396.136,Z 391.4,A -85,B 0,C 180,E1 -11242.355,E2 -11242.355} C_VEL
LIN {X 0,Y 395.948,Z 395.759,A -85,B 0,C 180,E1 -11243.888,E2 -11243.888} C_VEL
LIN {X 0,Y 395.92,Z 398.073,A -85,B 0,C 180,E1 -11244.91,E2 -11244.91} C_VEL
LIN {X 0,Y 395.802,Z 399.941,A -85,B 0,C 180,E1 -11245.929,E2 -11245.929} C_VEL
LIN {X 0,Y 395.811,Z 401.348,A -85,B 0,C 180,E1 -11246.948,E2 -11246.948} C_VEL
LIN {X 0,Y 395.854,Z 402.355,A -85,B 0,C 180,E1 -11247.967,E2 -11247.967} C_VEL
LIN {X 0,Y 395.812,Z 402.965,A -85,B 0,C 180,E1 -11248.984,E2 -11248.984} C_VEL
LIN {X 0,Y 395.815,Z 403.18,A -85,B 0,C 180,E1 -11250.001,E2 -11250.001} C_VEL
LIN {X 0,Y 395.854,Z 402.342,A -85,B 0,C 180,E1 -11252.036,E2 -11252.036} C_VEL
LIN {X 0,Y 395.813,Z 401.33,A -85,B 0,C 180,E1 -11253.055,E2 -11253.055} C_VEL
LIN {X 0,Y 395.802,Z 399.91,A -85,B 0,C 180,E1 -11254.074,E2 -11254.074} C_VEL
LIN {X 0,Y 395.908,Z 396.937,A -85,B 0,C 180,E1 -11255.604,E2 -11255.604} C_VEL
LIN {X 0,Y 396.063,Z 392.912,A -85,B 0,C 180,E1 -11257.137,E2 -11257.137} C_VEL
LIN {X 0,Y 396.459,Z 386.724,A -85,B 0,C 180,E1 -11258.925,E2 -11258.925} C_VEL
LIN {X 0,Y 396.918,Z 379.968,A -85,B 0,C 180,E1 -11260.458,E2 -11260.458} C_VEL
LIN {X 0,Y 397.598,Z 371.595,A -85,B 0,C 180,E1 -11261.989,E2 -11261.989} C_VEL
LIN {X 0,Y 398.286,Z 362.993,A -85,B 0,C 180,E1 -11263.263,E2 -11263.263} C_VEL
LIN {X 0,Y 399.105,Z 352.611,A -85,B 0,C 180,E1 -11264.508,E2 -11264.508} C_VEL
LIN {X 0,Y 399.905,Z 341.858,A -85,B 0,C 180,E1 -11265.547,E2 -11265.547} C_VEL
LIN {X 0,Y 400.784,Z 330.544,A -85,B 0,C 180,E1 -11266.41,E2 -11266.41} C_VEL
LIN {X 0,Y 400.993,Z 325.318,A -85,B 0,C 180,E1 -11266.744,E2 -11266.744} C_VEL
LIN {X 0,Y 399.264,Z 312.14,A -85,B 0,C 180,E1 -11267.496,E2 -11267.496} C_VEL
LIN {X 0,Y 397.04,Z 298.175,A -85,B 0,C 180,E1 -11268.077,E2 -11268.077} C_VEL
LIN {X 0,Y 396.594,Z 295.014,A -85,B 0,C 180,E1 -11268.201,E2 -11268.201} C_VEL
LIN {X 0,Y 397.04,Z 286.256,A -85,B 0,C 180,E1 -11271.823,E2 -11271.823} C_VEL
LIN {X 0,Y 397.628,Z 277.095,A -85,B 0,C 180,E1 -11275.655,E2 -11275.655} C_VEL
LIN {X 0,Y 398.152,Z 269.131,A -85,B 0,C 180,E1 -11279.041,E2 -11279.041} C_VEL
LIN {X 0,Y 398.76,Z 261.866,A -85,B 0,C 180,E1 -11282.222,E2 -11282.222} C_VEL
LIN {X 0,Y 399.328,Z 254.648,A -85,B 0,C 180,E1 -11285.507,E2 -11285.507} C_VEL
LIN {X 0,Y 399.108,Z 250.364,A -85,B 0,C 180,E1 -11287.588,E2 -11287.588} C_VEL
LIN {X 0,Y 398.057,Z 244.18,A -85,B 0,C 180,E1 -11290.79,E2 -11290.79} C_VEL
LIN {X 0,Y 397.108,Z 239.024,A -85,B 0,C 180,E1 -11293.649,E2 -11293.649} C_VEL
LIN {X 0,Y 397.109,Z 239.022,A -85,B 0,C 180,E1 -11296.522,E2 -11296.522} C_VEL
LIN {X 0,Y 397.119,Z 239.019,A -85,B 0,C 180,E1 -11300.423,E2 -11300.423} C_VEL
LIN {X 0,Y 397.112,Z 239.019,A -85,B 0,C 180,E1 -11304.266,E2 -11304.266} C_VEL
LIN {X 0,Y 397.118,Z 239.019,A -85,B 0,C 180,E1 -11306.727,E2 -11306.727} C_VEL
LIN {X 0,Y 397.124,Z 239.02,A -85,B 0,C 180,E1 -11310.296,E2 -11310.296} C_VEL
LIN {X 0,Y 397.11,Z 239.018,A -85,B 0,C 180,E1 -11313.74,E2 -11313.74} C_VEL
LIN {X 0,Y 397.116,Z 239.017,A -85,B 0,C 180,E1 -11317.086,E2 -11317.086} C_VEL
LIN {X 0,Y 397.153,Z 239.016,A -85,B 0,C 180,E1 -11320.353,E2 -11320.353} C_VEL
LIN {X 0,Y 397.134,Z 239.016,A -85,B 0,C 180,E1 -11323.552,E2 -11323.552} C_VEL
LIN {X 0,Y 397.237,Z 239.001,A -85,B 0,C 180,E1 -11326.703,E2 -11326.703} C_VEL
LIN {X 0,Y 397.213,Z 239.009,A -85,B 0,C 180,E1 -11329.809,E2 -11329.809} C_VEL
LIN {X 0,Y 397.341,Z 238.988,A -85,B 0,C 180,E1 -11332.888,E2 -11332.888} C_VEL
LIN {X 0,Y 397.257,Z 238.999,A -85,B 0,C 180,E1 -11334.925,E2 -11334.925} C_VEL
LIN {X 0,Y 397.456,Z 238.977,A -85,B 0,C 180,E1 -11337.973,E2 -11337.973} C_VEL
LIN {X 0,Y 397.582,Z 238.96,A -85,B 0,C 180,E1 -11340,E2 -11340} C_VEL
LIN {X 0,Y 397.343,Z 238.99,A -85,B 0,C 180,E1 -11343.042,E2 -11343.042} C_VEL
LIN {X 0,Y 397.297,Z 238.993,A -85,B 0,C 180,E1 -11346.519,E2 -11346.519} C_VEL
LIN {X 0,Y 397.238,Z 239.006,A -85,B 0,C 180,E1 -11349.162,E2 -11349.162} C_VEL
LIN {X 0,Y 397.226,Z 239.003,A -85,B 0,C 180,E1 -11352.258,E2 -11352.258} C_VEL
LIN {X 0,Y 397.187,Z 239.011,A -85,B 0,C 180,E1 -11355.392,E2 -11355.392} C_VEL
LIN {X 0,Y 397.166,Z 239.013,A -85,B 0,C 180,E1 -11358.573,E2 -11358.573} C_VEL
LIN {X 0,Y 397.102,Z 239.018,A -85,B 0,C 180,E1 -11361.818,E2 -11361.818} C_VEL
LIN {X 0,Y 397.109,Z 239.019,A -85,B 0,C 180,E1 -11365.135,E2 -11365.135} C_VEL
LIN {X 0,Y 397.069,Z 239.026,A -85,B 0,C 180,E1 -11368.548,E2 -11368.548} C_VEL
LIN {X 0,Y 397.089,Z 239.02,A -85,B 0,C 180,E1 -11371.836,E2 -11371.836} C_VEL
LIN {X 0,Y 397.132,Z 239.018,A -85,B 0,C 180,E1 -11374.493,E2 -11374.493} C_VEL
LIN {X 0,Y 397.106,Z 239.022,A -85,B 0,C 180,E1 -11378.275,E2 -11378.275} C_VEL
LIN {X 0,Y 397.094,Z 239.02,A -85,B 0,C 180,E1 -11380.908,E2 -11380.908} C_VEL
LIN {X 0,Y 397.107,Z 239.018,A -85,B 0,C 180,E1 -11383.648,E2 -11383.648} C_VEL
LIN {X 0,Y 397.097,Z 239.02,A -85,B 0,C 180,E1 -11386.522,E2 -11386.522} C_VEL
LIN {X 0,Y 397.093,Z 239.021,A -85,B 0,C 180,E1 -11390.419,E2 -11390.419} C_VEL
LIN {X 0,Y 397.103,Z 239.018,A -85,B 0,C 180,E1 -11393.004,E2 -11393.004} C_VEL
LIN {X 0,Y 397.1,Z 239.021,A -85,B 0,C 180,E1 -11396.287,E2 -11396.287} C_VEL
LIN {X 0,Y 396.93,Z 239.041,A -85,B 0,C 180,E1 -11399.103,E2 -11399.103} C_VEL
LIN {X 0,Y 396.566,Z 239.091,A -85,B 0,C 180,E1 -11402.561,E2 -11402.561} C_VEL
LIN {X 0,Y 396.498,Z 241.005,A -85,B 0,C 180,E1 -11404.822,E2 -11404.822} C_VEL
LIN {X 0,Y 396.358,Z 244.187,A -85,B 0,C 180,E1 -11408.137,E2 -11408.137} C_VEL
LIN {X 0,Y 396.29,Z 247.444,A -85,B 0,C 180,E1 -11411.383,E2 -11411.383} C_VEL
LIN {X 0,Y 396.327,Z 249.595,A -85,B 0,C 180,E1 -11413.516,E2 -11413.516} C_VEL
LIN {X 0,Y 396.293,Z 252.558,A -85,B 0,C 180,E1 -11416.165,E2 -11416.165} C_VEL
LIN {X 0,Y 399.674,Z 265.896,A -85,B 0,C 180,E1 -11416.784,E2 -11416.784} C_VEL
LIN {X 0,Y 401.461,Z 274.343,A -85,B 0,C 180,E1 -11417.278,E2 -11417.278} C_VEL
LIN {X 0,Y 401.205,Z 283.923,A -85,B 0,C 180,E1 -11417.864,E2 -11417.864} C_VEL
LIN {X 0,Y 400.505,Z 295.268,A -85,B 0,C 180,E1 -11418.741,E2 -11418.741} C_VEL
LIN {X 0,Y 399.754,Z 306.738,A -85,B 0,C 180,E1 -11419.873,E2 -11419.873} C_VEL
LIN {X 0,Y 399.047,Z 316.902,A -85,B 0,C 180,E1 -11421.134,E2 -11421.134} C_VEL
LIN {X 0,Y 398.313,Z 325.168,A -85,B 0,C 180,E1 -11422.394,E2 -11422.394} C_VEL
LIN {X 0,Y 397.566,Z 333.252,A -85,B 0,C 180,E1 -11423.91,E2 -11423.91} C_VEL
LIN {X 0,Y 397.012,Z 339.758,A -85,B 0,C 180,E1 -11425.43,E2 -11425.43} C_VEL
LIN {X 0,Y 396.5,Z 344.951,A -85,B 0,C 180,E1 -11426.95,E2 -11426.95} C_VEL
LIN {X 0,Y 396.202,Z 348.988,A -85,B 0,C 180,E1 -11428.474,E2 -11428.474} C_VEL
LIN {X 0,Y 396.051,Z 351.988,A -85,B 0,C 180,E1 -11429.999,E2 -11429.999} C_VEL
LIN {X 0,Y 395.982,Z 353.477,A -85,B 0,C 180,E1 -11431.015,E2 -11431.015} C_VEL
LIN {X 0,Y 396.058,Z 355.178,A -85,B 0,C 180,E1 -11433.05,E2 -11433.05} C_VEL
LIN {X 0,Y 395.983,Z 355.375,A -85,B 0,C 180,E1 -11435.09,E2 -11435.09} C_VEL
LIN {X 0,Y 396.073,Z 354.593,A -85,B 0,C 180,E1 -11436.444,E2 -11436.444} C_VEL
LIN {X 0,Y 396.171,Z 352.639,A -85,B 0,C 180,E1 -11438.157,E2 -11438.157} C_VEL
LIN {X 0,Y 396.414,Z 349.872,A -85,B 0,C 180,E1 -11439.695,E2 -11439.695} C_VEL
LIN {X 0,Y 396.696,Z 346.084,A -85,B 0,C 180,E1 -11441.236,E2 -11441.236} C_VEL
LIN {X 0,Y 397.209,Z 341.157,A -85,B 0,C 180,E1 -11442.776,E2 -11442.776} C_VEL
LIN {X 0,Y 397.829,Z 334.943,A -85,B 0,C 180,E1 -11444.317,E2 -11444.317} C_VEL
LIN {X 0,Y 398.602,Z 327.13,A -85,B 0,C 180,E1 -11445.858,E2 -11445.858} C_VEL
LIN {X 0,Y 399.352,Z 319.357,A -85,B 0,C 180,E1 -11447.108,E2 -11447.108} C_VEL
LIN {X 0,Y 399.058,Z 315.264,A -85,B 0,C 180,E1 -11447.716,E2 -11447.716} C_VEL
LIN {X 0,Y 396.889,Z 308.414,A -85,B 0,C 180,E1 -11448.702,E2 -11448.702} C_VEL
LIN {X 0,Y 394.791,Z 301.121,A -85,B 0,C 180,E1 -11449.617,E2 -11449.617} C_VEL
LIN {X 0,Y 394.599,Z 296.241,A -85,B 0,C 180,E1 -11450.104,E2 -11450.104} C_VEL
LIN {X 0,Y 395.438,Z 284.247,A -85,B 0,C 180,E1 -11451.053,E2 -11451.053} C_VEL
LIN {X 0,Y 395.745,Z 277.588,A -85,B 0,C 180,E1 -11451.476,E2 -11451.476} C_VEL
LIN {X 0,Y 392.9,Z 265.609,A -85,B 0,C 180,E1 -11452.26,E2 -11452.26} C_VEL
LIN {X 0,Y 389.239,Z 253.04,A -85,B 0,C 180,E1 -11452.93,E2 -11452.93} C_VEL
LIN {X 0,Y 389.333,Z 250.263,A -85,B 0,C 180,E1 -11455.671,E2 -11455.671} C_VEL
LIN {X 0,Y 389.465,Z 246.898,A -85,B 0,C 180,E1 -11459.156,E2 -11459.156} C_VEL
LIN {X 0,Y 389.512,Z 243.529,A -85,B 0,C 180,E1 -11462.77,E2 -11462.77} C_VEL
LIN {X 0,Y 389.672,Z 240.147,A -85,B 0,C 180,E1 -11466.523,E2 -11466.523} C_VEL
LIN {X 0,Y 389.927,Z 239.915,A -85,B 0,C 180,E1 -11469.192,E2 -11469.192} C_VEL
LIN {X 0,Y 390.032,Z 239.902,A -85,B 0,C 180,E1 -11472.372,E2 -11472.372} C_VEL
LIN {X 0,Y 390.037,Z 239.9,A -85,B 0,C 180,E1 -11475.353,E2 -11475.353} C_VEL
LIN {X 0,Y 390.02,Z 239.903,A -85,B 0,C 180,E1 -11478.185,E2 -11478.185} C_VEL
LIN {X 0,Y 390.081,Z 239.896,A -85,B 0,C 180,E1 -11480.906,E2 -11480.906} C_VEL
LIN {X 0,Y 390.077,Z 239.895,A -85,B 0,C 180,E1 -11484.792,E2 -11484.792} C_VEL
LIN {X 0,Y 390.014,Z 239.902,A -85,B 0,C 180,E1 -11488.494,E2 -11488.494} C_VEL
LIN {X 0,Y 390.107,Z 239.891,A -85,B 0,C 180,E1 -11492.069,E2 -11492.069} C_VEL
LIN {X 0,Y 390.07,Z 239.897,A -85,B 0,C 180,E1 -11495.518,E2 -11495.518} C_VEL
LIN {X 0,Y 390.045,Z 239.901,A -85,B 0,C 180,E1 -11498.877,E2 -11498.877} C_VEL
LIN {X 0,Y 390.117,Z 239.891,A -85,B 0,C 180,E1 -11502.166,E2 -11502.166} C_VEL
LIN {X 0,Y 390.133,Z 239.89,A -85,B 0,C 180,E1 -11505.392,E2 -11505.392} C_VEL
LIN {X 0,Y 390.135,Z 239.888,A -85,B 0,C 180,E1 -11508.571,E2 -11508.571} C_VEL
LIN {X 0,Y 390.333,Z 239.865,A -85,B 0,C 180,E1 -11511.993,E2 -11511.993} C_VEL
LIN {X 0,Y 390.225,Z 239.876,A -85,B 0,C 180,E1 -11514.833,E2 -11514.833} C_VEL
LIN {X 0,Y 390.41,Z 239.852,A -85,B 0,C 180,E1 -11517.937,E2 -11517.937} C_VEL
LIN {X 0,Y 390.535,Z 239.838,A -85,B 0,C 180,E1 -11520,E2 -11520} C_VEL
LIN {X 0,Y 390.306,Z 239.866,A -85,B 0,C 180,E1 -11523.096,E2 -11523.096} C_VEL
LIN {X 0,Y 390.33,Z 239.863,A -85,B 0,C 180,E1 -11526.202,E2 -11526.202} C_VEL
LIN {X 0,Y 390.303,Z 239.868,A -85,B 0,C 180,E1 -11528.282,E2 -11528.282} C_VEL
LIN {X 0,Y 390.159,Z 239.883,A -85,B 0,C 180,E1 -11532.483,E2 -11532.483} C_VEL
LIN {X 0,Y 390.128,Z 239.886,A -85,B 0,C 180,E1 -11535.677,E2 -11535.677} C_VEL
LIN {X 0,Y 390.094,Z 239.89,A -85,B 0,C 180,E1 -11538.923,E2 -11538.923} C_VEL
LIN {X 0,Y 390.029,Z 239.902,A -85,B 0,C 180,E1 -11542.235,E2 -11542.235} C_VEL
LIN {X 0,Y 390.109,Z 239.891,A -85,B 0,C 180,E1 -11545.744,E2 -11545.744} C_VEL
LIN {X 0,Y 390.055,Z 239.898,A -85,B 0,C 180,E1 -11549.11,E2 -11549.11} C_VEL
LIN {X 0,Y 390.046,Z 239.899,A -85,B 0,C 180,E1 -11552.721,E2 -11552.721} C_VEL
LIN {X 0,Y 390.046,Z 239.899,A -85,B 0,C 180,E1 -11555.826,E2 -11555.826} C_VEL
LIN {X 0,Y 390.06,Z 239.897,A -85,B 0,C 180,E1 -11559.219,E2 -11559.219} C_VEL
LIN {X 0,Y 390.031,Z 239.901,A -85,B 0,C 180,E1 -11562.375,E2 -11562.375} C_VEL
LIN {X 0,Y 390.044,Z 239.985,A -85,B 0,C 180,E1 -11564.929,E2 -11564.929} C_VEL
LIN {X 0,Y 391.133,Z 245.583,A -85,B 0,C 180,E1 -11568.333,E2 -11568.333} C_VEL
LIN {X 0,Y 391.993,Z 250.555,A -85,B 0,C 180,E1 -11571.135,E2 -11571.135} C_VEL
LIN {X 0,Y 392.566,Z 254.321,A -85,B 0,C 180,E1 -11573.145,E2 -11573.145} C_VEL
LIN {X 0,Y 392.36,Z 259.048,A -85,B 0,C 180,E1 -11575.483,E2 -11575.483} C_VEL
LIN {X 0,Y 391.632,Z 265.761,A -85,B 0,C 180,E1 -11578.642,E2 -11578.642} C_VEL
LIN {X 0,Y 390.997,Z 273.452,A -85,B 0,C 180,E1 -11582.14,E2 -11582.14} C_VEL
LIN {X 0,Y 390.353,Z 281.143,A -85,B 0,C 180,E1 -11585.539,E2 -11585.539} C_VEL
LIN {X 0,Y 389.917,Z 288.844,A -85,B 0,C 180,E1 -11588.872,E2 -11588.872} C_VEL
LIN {X 0,Y 389.559,Z 294.577,A -85,B 0,C 180,E1 -11591.325,E2 -11591.325} C_VEL
LIN {X 0,Y 391.996,Z 308.445,A -85,B 0,C 180,E1 -11591.893,E2 -11591.893} C_VEL
LIN {X 0,Y 393.59,Z 321.04,A -85,B 0,C 180,E1 -11592.594,E2 -11592.594} C_VEL
LIN {X 0,Y 394.259,Z 328.253,A -85,B 0,C 180,E1 -11593.08,E2 -11593.08} C_VEL
LIN {X 0,Y 393.339,Z 339.6,A -85,B 0,C 180,E1 -11593.924,E2 -11593.924} C_VEL
LIN {X 0,Y 392.426,Z 350.396,A -85,B 0,C 180,E1 -11594.95,E2 -11594.95} C_VEL
LIN {X 0,Y 391.627,Z 359.988,A -85,B 0,C 180,E1 -11596.081,E2 -11596.081} C_VEL
LIN {X 0,Y 390.797,Z 370.015,A -85,B 0,C 180,E1 -11597.539,E2 -11597.539} C_VEL
LIN {X 0,Y 389.982,Z 378.596,A -85,B 0,C 180,E1 -11599.094,E2 -11599.094} C_VEL
LIN {X 0,Y 389.451,Z 385.49,A -85,B 0,C 180,E1 -11600.655,E2 -11600.655} C_VEL
LIN {X 0,Y 389.075,Z 391.023,A -85,B 0,C 180,E1 -11602.215,E2 -11602.215} C_VEL
LIN {X 0,Y 388.831,Z 396.147,A -85,B 0,C 180,E1 -11604.098,E2 -11604.098} C_VEL
LIN {X 0,Y 388.729,Z 399.536,A -85,B 0,C 180,E1 -11605.854,E2 -11605.854} C_VEL
LIN {X 0,Y 388.769,Z 401.939,A -85,B 0,C 180,E1 -11607.93,E2 -11607.93} C_VEL
LIN {X 0,Y 388.743,Z 402.546,A -85,B 0,C 180,E1 -11608.966,E2 -11608.966} C_VEL
LIN {X 0,Y 388.742,Z 402.753,A -85,B 0,C 180,E1 -11610.002,E2 -11610.002} C_VEL
LIN {X 0,Y 388.788,Z 401.905,A -85,B 0,C 180,E1 -11612.073,E2 -11612.073} C_VEL
LIN {X 0,Y 388.718,Z 400.886,A -85,B 0,C 180,E1 -11613.111,E2 -11613.111} C_VEL
LIN {X 0,Y 388.729,Z 399.458,A -85,B 0,C 180,E1 -11614.149,E2 -11614.149} C_VEL
LIN {X 0,Y 388.833,Z 396.012,A -85,B 0,C 180,E1 -11615.903,E2 -11615.903} C_VEL
LIN {X 0,Y 389.079,Z 390.816,A -85,B 0,C 180,E1 -11617.787,E2 -11617.787} C_VEL
LIN {X 0,Y 389.454,Z 385.205,A -85,B 0,C 180,E1 -11619.348,E2 -11619.348} C_VEL
LIN {X 0,Y 389.969,Z 378.203,A -85,B 0,C 180,E1 -11620.909,E2 -11620.909} C_VEL
LIN {X 0,Y 390.779,Z 369.437,A -85,B 0,C 180,E1 -11622.465,E2 -11622.465} C_VEL
LIN {X 0,Y 391.527,Z 360.728,A -85,B 0,C 180,E1 -11623.724,E2 -11623.724} C_VEL
LIN {X 0,Y 392.264,Z 350.581,A -85,B 0,C 180,E1 -11624.926,E2 -11624.926} C_VEL
LIN {X 0,Y 393.141,Z 339.743,A -85,B 0,C 180,E1 -11625.955,E2 -11625.955} C_VEL
LIN {X 0,Y 394.004,Z 328.343,A -85,B 0,C 180,E1 -11626.8,E2 -11626.8} C_VEL
LIN {X 0,Y 393.724,Z 323.246,A -85,B 0,C 180,E1 -11627.136,E2 -11627.136} C_VEL
LIN {X 0,Y 391.936,Z 310.019,A -85,B 0,C 180,E1 -11627.883,E2 -11627.883} C_VEL
LIN {X 0,Y 389.937,Z 297.249,A -85,B 0,C 180,E1 -11628.408,E2 -11628.408} C_VEL
LIN {X 0,Y 389.543,Z 294.64,A -85,B 0,C 180,E1 -11628.502,E2 -11628.502} C_VEL
LIN {X 0,Y 389.932,Z 287.136,A -85,B 0,C 180,E1 -11631.685,E2 -11631.685} C_VEL
LIN {X 0,Y 390.532,Z 277.986,A -85,B 0,C 180,E1 -11635.59,E2 -11635.59} C_VEL
LIN {X 0,Y 391.121,Z 270.087,A -85,B 0,C 180,E1 -11639.024,E2 -11639.024} C_VEL
LIN {X 0,Y 391.688,Z 263.514,A -85,B 0,C 180,E1 -11641.944,E2 -11641.944} C_VEL
LIN {X 0,Y 392.266,Z 256.948,A -85,B 0,C 180,E1 -11644.984,E2 -11644.984} C_VEL
LIN {X 0,Y 392.297,Z 253.026,A -85,B 0,C 180,E1 -11646.882,E2 -11646.882} C_VEL
LIN {X 0,Y 391.555,Z 247.989,A -85,B 0,C 180,E1 -11649.484,E2 -11649.484} C_VEL
LIN {X 0,Y 390.569,Z 242.526,A -85,B 0,C 180,E1 -11652.459,E2 -11652.459} C_VEL
LIN {X 0,Y 390.045,Z 239.905,A -85,B 0,C 180,E1 -11654.098,E2 -11654.098} C_VEL
LIN {X 0,Y 390.049,Z 239.903,A -85,B 0,C 180,E1 -11657.627,E2 -11657.627} C_VEL
LIN {X 0,Y 390.094,Z 239.895,A -85,B 0,C 180,E1 -11660.908,E2 -11660.908} C_VEL
LIN {X 0,Y 390.088,Z 239.895,A -85,B 0,C 180,E1 -11664.793,E2 -11664.793} C_VEL
LIN {X 0,Y 390.029,Z 239.904,A -85,B 0,C 180,E1 -11668.496,E2 -11668.496} C_VEL
LIN {X 0,Y 390.082,Z 239.896,A -85,B 0,C 180,E1 -11672.067,E2 -11672.067} C_VEL
LIN {X 0,Y 390.07,Z 239.894,A -85,B 0,C 180,E1 -11675.519,E2 -11675.519} C_VEL
LIN {X 0,Y 390.063,Z 239.895,A -85,B 0,C 180,E1 -11678.878,E2 -11678.878} C_VEL
LIN {X 0,Y 390.11,Z 239.894,A -85,B 0,C 180,E1 -11682.166,E2 -11682.166} C_VEL
LIN {X 0,Y 390.098,Z 239.891,A -85,B 0,C 180,E1 -11685.391,E2 -11685.391} C_VEL
LIN {X 0,Y 390.174,Z 239.883,A -85,B 0,C 180,E1 -11687.517,E2 -11687.517} C_VEL
LIN {X 0,Y 390.195,Z 239.878,A -85,B 0,C 180,E1 -11690.671,E2 -11690.671} C_VEL
LIN {X 0,Y 390.324,Z 239.866,A -85,B 0,C 180,E1 -11693.798,E2 -11693.798} C_VEL
LIN {X 0,Y 390.425,Z 239.853,A -85,B 0,C 180,E1 -11697.937,E2 -11697.937} C_VEL
LIN {X 0,Y 390.552,Z 239.836,A -85,B 0,C 180,E1 -11700,E2 -11700} C_VEL
LIN {X 0,Y 390.28,Z 239.871,A -85,B 0,C 180,E1 -11703.097,E2 -11703.097} C_VEL
LIN {X 0,Y 390.257,Z 239.87,A -85,B 0,C 180,E1 -11706.512,E2 -11706.512} C_VEL
LIN {X 0,Y 390.197,Z 239.882,A -85,B 0,C 180,E1 -11709.329,E2 -11709.329} C_VEL
LIN {X 0,Y 390.178,Z 239.881,A -85,B 0,C 180,E1 -11712.483,E2 -11712.483} C_VEL
LIN {X 0,Y 390.147,Z 239.885,A -85,B 0,C 180,E1 -11715.677,E2 -11715.677} C_VEL
LIN {X 0,Y 390.111,Z 239.893,A -85,B 0,C 180,E1 -11718.922,E2 -11718.922} C_VEL
LIN {X 0,Y 390.042,Z 239.898,A -85,B 0,C 180,E1 -11722.234,E2 -11722.234} C_VEL
LIN {X 0,Y 390.058,Z 239.895,A -85,B 0,C 180,E1 -11725.722,E2 -11725.722} C_VEL
LIN {X 0,Y 390.031,Z 239.9,A -85,B 0,C 180,E1 -11729.112,E2 -11729.112} C_VEL
LIN {X 0,Y 390.051,Z 239.9,A -85,B 0,C 180,E1 -11732.721,E2 -11732.721} C_VEL
LIN {X 0,Y 390.063,Z 239.896,A -85,B 0,C 180,E1 -11735.825,E2 -11735.825} C_VEL
LIN {X 0,Y 390.069,Z 239.894,A -85,B 0,C 180,E1 -11739.216,E2 -11739.216} C_VEL
LIN {X 0,Y 390.047,Z 239.902,A -85,B 0,C 180,E1 -11742.373,E2 -11742.373} C_VEL
LIN {X 0,Y 390.047,Z 239.896,A -85,B 0,C 180,E1 -11745.353,E2 -11745.353} C_VEL
LIN {X 0,Y 390.02,Z 239.904,A -85,B 0,C 180,E1 -11748.184,E2 -11748.184} C_VEL
LIN {X 0,Y 390.064,Z 239.894,A -85,B 0,C 180,E1 -11750.903,E2 -11750.903} C_VEL
LIN {X 0,Y 390.075,Z 239.893,A -85,B 0,C 180,E1 -11754.791,E2 -11754.791} C_VEL
LIN {X 0,Y 389.987,Z 239.909,A -85,B 0,C 180,E1 -11757.887,E2 -11757.887} C_VEL
LIN {X 0,Y 389.696,Z 239.941,A -85,B 0,C 180,E1 -11760.859,E2 -11760.859} C_VEL
LIN {X 0,Y 389.46,Z 240.285,A -85,B 0,C 180,E1 -11763.182,E2 -11763.182} C_VEL
LIN {X 0,Y 389.351,Z 243.516,A -85,B 0,C 180,E1 -11766.601,E2 -11766.601} C_VEL
LIN {X 0,Y 389.281,Z 246.767,A -85,B 0,C 180,E1 -11769.937,E2 -11769.937} C_VEL
LIN {X 0,Y 389.275,Z 250.038,A -85,B 0,C 180,E1 -11773.209,E2 -11773.209} C_VEL
LIN {X 0,Y 389.213,Z 252.804,A -85,B 0,C 180,E1 -11775.839,E2 -11775.839} C_VEL
LIN {X 0,Y 392.907,Z 267.432,A -85,B 0,C 180,E1 -11776.552,E2 -11776.552} C_VEL
LIN {X 0,Y 394.638,Z 275.705,A -85,B 0,C 180,E1 -11777.06,E2 -11777.06} C_VEL
LIN {X 0,Y 394.325,Z 285.018,A -85,B 0,C 180,E1 -11777.649,E2 -11777.649} C_VEL
LIN {X 0,Y 393.605,Z 296.223,A -85,B 0,C 180,E1 -11778.541,E2 -11778.541} C_VEL
LIN {X 0,Y 392.835,Z 307.598,A -85,B 0,C 180,E1 -11779.693,E2 -11779.693} C_VEL
LIN {X 0,Y 392.083,Z 317.66,A -85,B 0,C 180,E1 -11780.975,E2 -11780.975} C_VEL
LIN {X 0,Y 391.329,Z 325.87,A -85,B 0,C 180,E1 -11782.258,E2 -11782.258} C_VEL
LIN {X 0,Y 390.558,Z 333.906,A -85,B 0,C 180,E1 -11783.8,E2 -11783.8} C_VEL
LIN {X 0,Y 389.974,Z 340.371,A -85,B 0,C 180,E1 -11785.347,E2 -11785.347} C_VEL
LIN {X 0,Y 389.445,Z 345.527,A -85,B 0,C 180,E1 -11786.895,E2 -11786.895} C_VEL
LIN {X 0,Y 389.143,Z 349.53,A -85,B 0,C 180,E1 -11788.446,E2 -11788.446} C_VEL
LIN {X 0,Y 388.965,Z 352.499,A -85,B 0,C 180,E1 -11789.998,E2 -11789.998} C_VEL
LIN {X 0,Y 388.904,Z 353.96,A -85,B 0,C 180,E1 -11791.034,E2 -11791.034} C_VEL
LIN {X 0,Y 388.972,Z 355.627,A -85,B 0,C 180,E1 -11793.106,E2 -11793.106} C_VEL
LIN {X 0,Y 388.863,Z 355.907,A -85,B 0,C 180,E1 -11794.144,E2 -11794.144} C_VEL
LIN {X 0,Y 388.923,Z 355.784,A -85,B 0,C 180,E1 -11795.182,E2 -11795.182} C_VEL
LIN {X 0,Y 389.009,Z 355.062,A -85,B 0,C 180,E1 -11796.456,E2 -11796.456} C_VEL
LIN {X 0,Y 389.127,Z 352.998,A -85,B 0,C 180,E1 -11798.306,E2 -11798.306} C_VEL
LIN {X 0,Y 389.373,Z 350.201,A -85,B 0,C 180,E1 -11799.872,E2 -11799.872} C_VEL
LIN {X 0,Y 389.703,Z 346.379,A -85,B 0,C 180,E1 -11801.44,E2 -11801.44} C_VEL
LIN {X 0,Y 390.24,Z 341.415,A -85,B 0,C 180,E1 -11803.008,E2 -11803.008} C_VEL
LIN {X 0,Y 390.909,Z 335.155,A -85,B 0,C 180,E1 -11804.576,E2 -11804.576} C_VEL
LIN {X 0,Y 391.742,Z 327.278,A -85,B 0,C 180,E1 -11806.144,E2 -11806.144} C_VEL
LIN {X 0,Y 392.548,Z 319.224,A -85,B 0,C 180,E1 -11807.449,E2 -11807.449} C_VEL
LIN {X 0,Y 393.556,Z 308.694,A -85,B 0,C 180,E1 -11808.833,E2 -11808.833} C_VEL
LIN {X 0,Y 394.456,Z 298.254,A -85,B 0,C 180,E1 -11809.921,E2 -11809.921} C_VEL
LIN {X 0,Y 394.599,Z 296.241,A -85,B 0,C 180,E1 -11810.104,E2 -11810.104} C_VEL
LIN {X 0,Y 394.38,Z 291.232,A -85,B 0,C 180,E1 -11810.564,E2 -11810.564} C_VEL
LIN {X 0,Y 393.125,Z 286.322,A -85,B 0,C 180,E1 -11811.022,E2 -11811.022} C_VEL
LIN {X 0,Y 389.229,Z 276.54,A -85,B 0,C 180,E1 -11811.893,E2 -11811.893} C_VEL
LIN {X 0,Y 386.877,Z 269.636,A -85,B 0,C 180,E1 -11812.408,E2 -11812.408} C_VEL
LIN {X 0,Y 383.383,Z 257.633,A -85,B 0,C 180,E1 -11813.107,E2 -11813.107} C_VEL
LIN {X 0,Y 382.209,Z 253.45,A -85,B 0,C 180,E1 -11813.336,E2 -11813.336} C_VEL
LIN {X 0,Y 382.28,Z 250.613,A -85,B 0,C 180,E1 -11816.18,E2 -11816.18} C_VEL
LIN {X 0,Y 382.37,Z 248.355,A -85,B 0,C 180,E1 -11818.545,E2 -11818.545} C_VEL
LIN {X 0,Y 382.437,Z 246.074,A -85,B 0,C 180,E1 -11820.966,E2 -11820.966} C_VEL
LIN {X 0,Y 382.546,Z 242.682,A -85,B 0,C 180,E1 -11824.715,E2 -11824.715} C_VEL
LIN {X 0,Y 382.615,Z 241.471,A -85,B 0,C 180,E1 -11826.078,E2 -11826.078} C_VEL
LIN {X 0,Y 382.803,Z 240.803,A -85,B 0,C 180,E1 -11827.865,E2 -11827.865} C_VEL
LIN {X 0,Y 382.954,Z 240.783,A -85,B 0,C 180,E1 -11831.349,E2 -11831.349} C_VEL
LIN {X 0,Y 382.989,Z 240.78,A -85,B 0,C 180,E1 -11834.302,E2 -11834.302} C_VEL
LIN {X 0,Y 383.003,Z 240.778,A -85,B 0,C 180,E1 -11837.239,E2 -11837.239} C_VEL
LIN {X 0,Y 383.006,Z 240.776,A -85,B 0,C 180,E1 -11840.412,E2 -11840.412} C_VEL
LIN {X 0,Y 383.018,Z 240.774,A -85,B 0,C 180,E1 -11844.043,E2 -11844.043} C_VEL
LIN {X 0,Y 382.977,Z 240.783,A -85,B 0,C 180,E1 -11847.577,E2 -11847.577} C_VEL
LIN {X 0,Y 382.982,Z 240.778,A -85,B 0,C 180,E1 -11850.299,E2 -11850.299} C_VEL
LIN {X 0,Y 383.07,Z 240.769,A -85,B 0,C 180,E1 -11854.02,E2 -11854.02} C_VEL
LIN {X 0,Y 382.998,Z 240.779,A -85,B 0,C 180,E1 -11857.334,E2 -11857.334} C_VEL
LIN {X 0,Y 383.05,Z 240.774,A -85,B 0,C 180,E1 -11860.716,E2 -11860.716} C_VEL
LIN {X 0,Y 383.07,Z 240.77,A -85,B 0,C 180,E1 -11864.026,E2 -11864.026} C_VEL
LIN {X 0,Y 383.125,Z 240.764,A -85,B 0,C 180,E1 -11867.283,E2 -11867.283} C_VEL
LIN {X 0,Y 383.248,Z 240.745,A -85,B 0,C 180,E1 -11871.564,E2 -11871.564} C_VEL
LIN {X 0,Y 383.286,Z 240.742,A -85,B 0,C 180,E1 -11873.684,E2 -11873.684} C_VEL
LIN {X 0,Y 383.377,Z 240.728,A -85,B 0,C 180,E1 -11877.899,E2 -11877.899} C_VEL
LIN {X 0,Y 383.504,Z 240.714,A -85,B 0,C 180,E1 -11880,E2 -11880} C_VEL
LIN {X 0,Y 383.242,Z 240.746,A -85,B 0,C 180,E1 -11883.154,E2 -11883.154} C_VEL
LIN {X 0,Y 383.285,Z 240.74,A -85,B 0,C 180,E1 -11886.316,E2 -11886.316} C_VEL
LIN {X 0,Y 383.248,Z 240.747,A -85,B 0,C 180,E1 -11888.436,E2 -11888.436} C_VEL
LIN {X 0,Y 383.085,Z 240.766,A -85,B 0,C 180,E1 -11891.642,E2 -11891.642} C_VEL
LIN {X 0,Y 383.098,Z 240.764,A -85,B 0,C 180,E1 -11894.882,E2 -11894.882} C_VEL
LIN {X 0,Y 383.078,Z 240.767,A -85,B 0,C 180,E1 -11898.173,E2 -11898.173} C_VEL
LIN {X 0,Y 382.985,Z 240.779,A -85,B 0,C 180,E1 -11901.531,E2 -11901.531} C_VEL
LIN {X 0,Y 383.041,Z 240.773,A -85,B 0,C 180,E1 -11904.961,E2 -11904.961} C_VEL
LIN {X 0,Y 383.039,Z 240.774,A -85,B 0,C 180,E1 -11908.493,E2 -11908.493} C_VEL
LIN {X 0,Y 382.998,Z 240.777,A -85,B 0,C 180,E1 -11912.428,E2 -11912.428} C_VEL
LIN {X 0,Y 383.015,Z 240.775,A -85,B 0,C 180,E1 -11915.957,E2 -11915.957} C_VEL
LIN {X 0,Y 383.006,Z 240.775,A -85,B 0,C 180,E1 -11919.588,E2 -11919.588} C_VEL
LIN {X 0,Y 382.997,Z 240.777,A -85,B 0,C 180,E1 -11922.78,E2 -11922.78} C_VEL
LIN {X 0,Y 383.01,Z 240.905,A -85,B 0,C 180,E1 -11924.491,E2 -11924.491} C_VEL
LIN {X 0,Y 384.099,Z 246.581,A -85,B 0,C 180,E1 -11928.036,E2 -11928.036} C_VEL
LIN {X 0,Y 384.992,Z 251.65,A -85,B 0,C 180,E1 -11930.967,E2 -11930.967} C_VEL
LIN {X 0,Y 385.591,Z 255.982,A -85,B 0,C 180,E1 -11933.319,E2 -11933.319} C_VEL
LIN {X 0,Y 385.176,Z 261.733,A -85,B 0,C 180,E1 -11936.187,E2 -11936.187} C_VEL
LIN {X 0,Y 384.346,Z 269.349,A -85,B 0,C 180,E1 -11939.813,E2 -11939.813} C_VEL
LIN {X 0,Y 383.863,Z 275.752,A -85,B 0,C 180,E1 -11942.762,E2 -11942.762} C_VEL
LIN {X 0,Y 383.148,Z 284.099,A -85,B 0,C 180,E1 -11946.512,E2 -11946.512} C_VEL
LIN {X 0,Y 382.659,Z 292.319,A -85,B 0,C 180,E1 -11950.139,E2 -11950.139} C_VEL
LIN {X 0,Y 382.54,Z 294.162,A -85,B 0,C 180,E1 -11950.944,E2 -11950.944} C_VEL
LIN {X 0,Y 385.019,Z 307.946,A -85,B 0,C 180,E1 -11951.525,E2 -11951.525} C_VEL
LIN {X 0,Y 386.69,Z 321.361,A -85,B 0,C 180,E1 -11952.294,E2 -11952.294} C_VEL
LIN {X 0,Y 387.426,Z 328.308,A -85,B 0,C 180,E1 -11952.782,E2 -11952.782} C_VEL
LIN {X 0,Y 386.523,Z 339.435,A -85,B 0,C 180,E1 -11953.632,E2 -11953.632} C_VEL
LIN {X 0,Y 385.547,Z 350.164,A -85,B 0,C 180,E1 -11954.675,E2 -11954.675} C_VEL
LIN {X 0,Y 384.672,Z 360.124,A -85,B 0,C 180,E1 -11955.88,E2 -11955.88} C_VEL
LIN {X 0,Y 383.847,Z 369.717,A -85,B 0,C 180,E1 -11957.31,E2 -11957.31} C_VEL
LIN {X 0,Y 382.974,Z 378.263,A -85,B 0,C 180,E1 -11958.892,E2 -11958.892} C_VEL
LIN {X 0,Y 382.426,Z 385.138,A -85,B 0,C 180,E1 -11960.481,E2 -11960.481} C_VEL
LIN {X 0,Y 382.012,Z 390.653,A -85,B 0,C 180,E1 -11962.071,E2 -11962.071} C_VEL
LIN {X 0,Y 381.803,Z 395.129,A -85,B 0,C 180,E1 -11963.721,E2 -11963.721} C_VEL
LIN {X 0,Y 381.733,Z 397.285,A -85,B 0,C 180,E1 -11964.72,E2 -11964.72} C_VEL
LIN {X 0,Y 381.657,Z 399.136,A -85,B 0,C 180,E1 -11965.777,E2 -11965.777} C_VEL
LIN {X 0,Y 381.687,Z 401.526,A -85,B 0,C 180,E1 -11967.891,E2 -11967.891} C_VEL
LIN {X 0,Y 381.675,Z 402.129,A -85,B 0,C 180,E1 -11968.946,E2 -11968.946} C_VEL
LIN {X 0,Y 381.672,Z 402.325,A -85,B 0,C 180,E1 -11970.002,E2 -11970.002} C_VEL
LIN {X 0,Y 381.676,Z 402.09,A -85,B 0,C 180,E1 -11971.057,E2 -11971.057} C_VEL
LIN {X 0,Y 381.704,Z 401.464,A -85,B 0,C 180,E1 -11972.112,E2 -11972.112} C_VEL
LIN {X 0,Y 381.625,Z 400.438,A -85,B 0,C 180,E1 -11973.169,E2 -11973.169} C_VEL
LIN {X 0,Y 381.658,Z 399.001,A -85,B 0,C 180,E1 -11974.226,E2 -11974.226} C_VEL
LIN {X 0,Y 381.735,Z 395.91,A -85,B 0,C 180,E1 -11975.856,E2 -11975.856} C_VEL
LIN {X 0,Y 381.929,Z 391.953,A -85,B 0,C 180,E1 -11977.402,E2 -11977.402} C_VEL
LIN {X 0,Y 382.334,Z 385.721,A -85,B 0,C 180,E1 -11979.257,E2 -11979.257} C_VEL
LIN {X 0,Y 382.844,Z 378.928,A -85,B 0,C 180,E1 -11980.847,E2 -11980.847} C_VEL
LIN {X 0,Y 383.646,Z 370.509,A -85,B 0,C 180,E1 -11982.432,E2 -11982.432} C_VEL
LIN {X 0,Y 384.431,Z 361.837,A -85,B 0,C 180,E1 -11983.75,E2 -11983.75} C_VEL
LIN {X 0,Y 385.276,Z 351.143,A -85,B 0,C 180,E1 -11985.068,E2 -11985.068} C_VEL
LIN {X 0,Y 386.144,Z 340.544,A -85,B 0,C 180,E1 -11986.116,E2 -11986.116} C_VEL
LIN {X 0,Y 387.082,Z 329.312,A -85,B 0,C 180,E1 -11986.991,E2 -11986.991} C_VEL
LIN {X 0,Y 386.897,Z 324.764,A -85,B 0,C 180,E1 -11987.305,E2 -11987.305} C_VEL
LIN {X 0,Y 385.179,Z 311.687,A -85,B 0,C 180,E1 -11988.09,E2 -11988.09} C_VEL
LIN {X 0,Y 383.153,Z 298.438,A -85,B 0,C 180,E1 -11988.672,E2 -11988.672} C_VEL
LIN {X 0,Y 382.514,Z 294.25,A -85,B 0,C 180,E1 -11988.826,E2 -11988.826} C_VEL
LIN {X 0,Y 382.91,Z 286.695,A -85,B 0,C 180,E1 -11992.104,E2 -11992.104} C_VEL
LIN {X 0,Y 383.579,Z 277.487,A -85,B 0,C 180,E1 -11996.131,E2 -11996.131} C_VEL
LIN {X 0,Y 384.137,Z 269.703,A -85,B 0,C 180,E1 -11999.604,E2 -11999.604} C_VEL
LIN {X 0,Y 384.813,Z 262.605,A -85,B 0,C 180,E1 -12002.847,E2 -12002.847} C_VEL
LIN {X 0,Y 385.339,Z 256.613,A -85,B 0,C 180,E1 -12005.708,E2 -12005.708} C_VEL
LIN {X 0,Y 385.15,Z 252.793,A -85,B 0,C 180,E1 -12007.633,E2 -12007.633} C_VEL
LIN {X 0,Y 384.26,Z 247.461,A -85,B 0,C 180,E1 -12010.489,E2 -12010.489} C_VEL
LIN {X 0,Y 383.224,Z 242.042,A -85,B 0,C 180,E1 -12013.579,E2 -12013.579} C_VEL
LIN {X 0,Y 383.021,Z 240.779,A -85,B 0,C 180,E1 -12014.398,E2 -12014.398} C_VEL
LIN {X 0,Y 383.017,Z 240.779,A -85,B 0,C 180,E1 -12017.241,E2 -12017.241} C_VEL
LIN {X 0,Y 383.02,Z 240.775,A -85,B 0,C 180,E1 -12020.415,E2 -12020.415} C_VEL
LIN {X 0,Y 383.029,Z 240.771,A -85,B 0,C 180,E1 -12024.045,E2 -12024.045} C_VEL
LIN {X 0,Y 382.991,Z 240.775,A -85,B 0,C 180,E1 -12027.579,E2 -12027.579} C_VEL
LIN {X 0,Y 382.991,Z 240.781,A -85,B 0,C 180,E1 -12030.3,E2 -12030.3} C_VEL
LIN {X 0,Y 383.05,Z 240.772,A -85,B 0,C 180,E1 -12034.033,E2 -12034.033} C_VEL
LIN {X 0,Y 383.004,Z 240.774,A -85,B 0,C 180,E1 -12037.335,E2 -12037.335} C_VEL
LIN {X 0,Y 383.063,Z 240.767,A -85,B 0,C 180,E1 -12040.716,E2 -12040.716} C_VEL
LIN {X 0,Y 383.027,Z 240.777,A -85,B 0,C 180,E1 -12044.024,E2 -12044.024} C_VEL
LIN {X 0,Y 383.141,Z 240.757,A -85,B 0,C 180,E1 -12047.284,E2 -12047.284} C_VEL
LIN {X 0,Y 383.145,Z 240.757,A -85,B 0,C 180,E1 -12050.498,E2 -12050.498} C_VEL
LIN {X 0,Y 383.279,Z 240.744,A -85,B 0,C 180,E1 -12053.684,E2 -12053.684} C_VEL
LIN {X 0,Y 383.392,Z 240.729,A -85,B 0,C 180,E1 -12057.899,E2 -12057.899} C_VEL
LIN {X 0,Y 383.521,Z 240.711,A -85,B 0,C 180,E1 -12060,E2 -12060} C_VEL
LIN {X 0,Y 383.217,Z 240.751,A -85,B 0,C 180,E1 -12063.154,E2 -12063.154} C_VEL
LIN {X 0,Y 383.222,Z 240.746,A -85,B 0,C 180,E1 -12066.501,E2 -12066.501} C_VEL
LIN {X 0,Y 383.148,Z 240.759,A -85,B 0,C 180,E1 -12069.502,E2 -12069.502} C_VEL
LIN {X 0,Y 383.134,Z 240.76,A -85,B 0,C 180,E1 -12073.536,E2 -12073.536} C_VEL
LIN {X 0,Y 383.102,Z 240.766,A -85,B 0,C 180,E1 -12077.069,E2 -12077.069} C_VEL
LIN {X 0,Y 383.037,Z 240.773,A -85,B 0,C 180,E1 -12080.647,E2 -12080.647} C_VEL
LIN {X 0,Y 383.015,Z 240.772,A -85,B 0,C 180,E1 -12083.809,E2 -12083.809} C_VEL
LIN {X 0,Y 382.974,Z 240.778,A -85,B 0,C 180,E1 -12087.309,E2 -12087.309} C_VEL
LIN {X 0,Y 382.989,Z 240.779,A -85,B 0,C 180,E1 -12090.918,E2 -12090.918} C_VEL
LIN {X 0,Y 383.026,Z 240.776,A -85,B 0,C 180,E1 -12094.667,E2 -12094.667} C_VEL
LIN {X 0,Y 383.005,Z 240.776,A -85,B 0,C 180,E1 -12097.903,E2 -12097.903} C_VEL
LIN {X 0,Y 382.989,Z 240.776,A -85,B 0,C 180,E1 -12101.347,E2 -12101.347} C_VEL
LIN {X 0,Y 383.002,Z 240.779,A -85,B 0,C 180,E1 -12104.302,E2 -12104.302} C_VEL
LIN {X 0,Y 382.989,Z 240.775,A -85,B 0,C 180,E1 -12107.235,E2 -12107.235} C_VEL
LIN {X 0,Y 382.992,Z 240.777,A -85,B 0,C 180,E1 -12110.418,E2 -12110.418} C_VEL
LIN {X 0,Y 383.021,Z 240.776,A -85,B 0,C 180,E1 -12114.042,E2 -12114.042} C_VEL
LIN {X 0,Y 382.991,Z 240.776,A -85,B 0,C 180,E1 -12116.596,E2 -12116.596} C_VEL
LIN {X 0,Y 382.784,Z 240.807,A -85,B 0,C 180,E1 -12119.648,E2 -12119.648} C_VEL
LIN {X 0,Y 382.431,Z 240.851,A -85,B 0,C 180,E1 -12122.648,E2 -12122.648} C_VEL
LIN {X 0,Y 382.348,Z 242.814,A -85,B 0,C 180,E1 -12124.989,E2 -12124.989} C_VEL
LIN {X 0,Y 382.253,Z 246.083,A -85,B 0,C 180,E1 -12128.424,E2 -12128.424} C_VEL
LIN {X 0,Y 382.176,Z 249.372,A -85,B 0,C 180,E1 -12131.781,E2 -12131.781} C_VEL
LIN {X 0,Y 382.188,Z 251.623,A -85,B 0,C 180,E1 -12133.987,E2 -12133.987} C_VEL
LIN {X 0,Y 382.147,Z 253.233,A -85,B 0,C 180,E1 -12135.512,E2 -12135.512} C_VEL
LIN {X 0,Y 385.974,Z 268.179,A -85,B 0,C 180,E1 -12136.269,E2 -12136.269} C_VEL
LIN {X 0,Y 387.81,Z 277.007,A -85,B 0,C 180,E1 -12136.831,E2 -12136.831} C_VEL
LIN {X 0,Y 387.367,Z 287.84,A -85,B 0,C 180,E1 -12137.557,E2 -12137.557} C_VEL
LIN {X 0,Y 386.608,Z 298.584,A -85,B 0,C 180,E1 -12138.464,E2 -12138.464} C_VEL
LIN {X 0,Y 385.825,Z 309.442,A -85,B 0,C 180,E1 -12139.624,E2 -12139.624} C_VEL
LIN {X 0,Y 385.12,Z 318.414,A -85,B 0,C 180,E1 -12140.81,E2 -12140.81} C_VEL
LIN {X 0,Y 384.347,Z 326.569,A -85,B 0,C 180,E1 -12142.116,E2 -12142.116} C_VEL
LIN {X 0,Y 383.553,Z 334.559,A -85,B 0,C 180,E1 -12143.687,E2 -12143.687} C_VEL
LIN {X 0,Y 382.921,Z 340.985,A -85,B 0,C 180,E1 -12145.261,E2 -12145.261} C_VEL
LIN {X 0,Y 382.379,Z 346.101,A -85,B 0,C 180,E1 -12146.838,E2 -12146.838} C_VEL
LIN {X 0,Y 382.086,Z 350.069,A -85,B 0,C 180,E1 -12148.417,E2 -12148.417} C_VEL
LIN {X 0,Y 381.883,Z 353.008,A -85,B 0,C 180,E1 -12149.998,E2 -12149.998} C_VEL
LIN {X 0,Y 381.828,Z 354.439,A -85,B 0,C 180,E1 -12151.053,E2 -12151.053} C_VEL
LIN {X 0,Y 381.889,Z 356.077,A -85,B 0,C 180,E1 -12153.163,E2 -12153.163} C_VEL
LIN {X 0,Y 381.783,Z 356.341,A -85,B 0,C 180,E1 -12154.221,E2 -12154.221} C_VEL
LIN {X 0,Y 381.865,Z 356.189,A -85,B 0,C 180,E1 -12155.278,E2 -12155.278} C_VEL
LIN {X 0,Y 381.928,Z 355.55,A -85,B 0,C 180,E1 -12156.445,E2 -12156.445} C_VEL
LIN {X 0,Y 382.069,Z 353.359,A -85,B 0,C 180,E1 -12158.461,E2 -12158.461} C_VEL
LIN {X 0,Y 382.349,Z 350.53,A -85,B 0,C 180,E1 -12160.055,E2 -12160.055} C_VEL
LIN {X 0,Y 382.721,Z 346.674,A -85,B 0,C 180,E1 -12161.652,E2 -12161.652} C_VEL
LIN {X 0,Y 383.26,Z 341.733,A -85,B 0,C 180,E1 -12163.232,E2 -12163.232} C_VEL
LIN {X 0,Y 383.972,Z 335.362,A -85,B 0,C 180,E1 -12164.846,E2 -12164.846} C_VEL
LIN {X 0,Y 384.877,Z 327.429,A -85,B 0,C 180,E1 -12166.44,E2 -12166.44} C_VEL
LIN {X 0,Y 385.745,Z 319.32,A -85,B 0,C 180,E1 -12167.767,E2 -12167.767} C_VEL
LIN {X 0,Y 386.73,Z 309.397,A -85,B 0,C 180,E1 -12169.092,E2 -12169.092} C_VEL
LIN {X 0,Y 387.615,Z 299.575,A -85,B 0,C 180,E1 -12170.149,E2 -12170.149} C_VEL
LIN {X 0,Y 388.501,Z 288.86,A -85,B 0,C 180,E1 -12171.07,E2 -12171.07} C_VEL
LIN {X 0,Y 388.939,Z 278.23,A -85,B 0,C 180,E1 -12171.806,E2 -12171.806} C_VEL
LIN {X 0,Y 386.877,Z 269.636,A -85,B 0,C 180,E1 -12172.408,E2 -12172.408} C_VEL
LIN {X 0,Y 385.354,Z 266.322,A -85,B 0,C 180,E1 -12172.667,E2 -12172.667} C_VEL
LIN {X 0,Y 382.969,Z 263.494,A -85,B 0,C 180,E1 -12172.929,E2 -12172.929} C_VEL
LIN {X 0,Y 376.878,Z 257.274,A -85,B 0,C 180,E1 -12173.503,E2 -12173.503} C_VEL
LIN {X 0,Y 375.17,Z 254.089,A -85,B 0,C 180,E1 -12173.71,E2 -12173.71} C_VEL
LIN {X 0,Y 375.229,Z 250.964,A -85,B 0,C 180,E1 -12176.711,E2 -12176.711} C_VEL
LIN {X 0,Y 375.356,Z 248.682,A -85,B 0,C 180,E1 -12179.129,E2 -12179.129} C_VEL
LIN {X 0,Y 375.449,Z 245.24,A -85,B 0,C 180,E1 -12182.876,E2 -12182.876} C_VEL
LIN {X 0,Y 375.602,Z 242.125,A -85,B 0,C 180,E1 -12186.429,E2 -12186.429} C_VEL
LIN {X 0,Y 375.589,Z 241.826,A -85,B 0,C 180,E1 -12186.78,E2 -12186.78} C_VEL
LIN {X 0,Y 375.837,Z 241.67,A -85,B 0,C 180,E1 -12189.476,E2 -12189.476} C_VEL
LIN {X 0,Y 375.919,Z 241.66,A -85,B 0,C 180,E1 -12192.3,E2 -12192.3} C_VEL
LIN {X 0,Y 375.92,Z 241.659,A -85,B 0,C 180,E1 -12195.267,E2 -12195.267} C_VEL
LIN {X 0,Y 375.925,Z 241.658,A -85,B 0,C 180,E1 -12198.398,E2 -12198.398} C_VEL
LIN {X 0,Y 375.966,Z 241.652,A -85,B 0,C 180,E1 -12201.728,E2 -12201.728} C_VEL
LIN {X 0,Y 375.971,Z 241.652,A -85,B 0,C 180,E1 -12205.331,E2 -12205.331} C_VEL
LIN {X 0,Y 375.948,Z 241.654,A -85,B 0,C 180,E1 -12208.437,E2 -12208.437} C_VEL
LIN {X 0,Y 375.974,Z 241.652,A -85,B 0,C 180,E1 -12212.139,E2 -12212.139} C_VEL
LIN {X 0,Y 375.996,Z 241.649,A -85,B 0,C 180,E1 -12214.538,E2 -12214.538} C_VEL
LIN {X 0,Y 375.953,Z 241.654,A -85,B 0,C 180,E1 -12218.045,E2 -12218.045} C_VEL
LIN {X 0,Y 375.998,Z 241.647,A -85,B 0,C 180,E1 -12221.472,E2 -12221.472} C_VEL
LIN {X 0,Y 376.047,Z 241.642,A -85,B 0,C 180,E1 -12224.832,E2 -12224.832} C_VEL
LIN {X 0,Y 376.037,Z 241.643,A -85,B 0,C 180,E1 -12228.136,E2 -12228.136} C_VEL
LIN {X 0,Y 376.247,Z 241.618,A -85,B 0,C 180,E1 -12231.876,E2 -12231.876} C_VEL
LIN {X 0,Y 376.169,Z 241.627,A -85,B 0,C 180,E1 -12234.64,E2 -12234.64} C_VEL
LIN {X 0,Y 376.343,Z 241.605,A -85,B 0,C 180,E1 -12237.859,E2 -12237.859} C_VEL
LIN {X 0,Y 376.474,Z 241.59,A -85,B 0,C 180,E1 -12240,E2 -12240} C_VEL
LIN {X 0,Y 376.181,Z 241.626,A -85,B 0,C 180,E1 -12243.213,E2 -12243.213} C_VEL
LIN {X 0,Y 376.243,Z 241.618,A -85,B 0,C 180,E1 -12246.435,E2 -12246.435} C_VEL
LIN {X 0,Y 376.193,Z 241.626,A -85,B 0,C 180,E1 -12248.595,E2 -12248.595} C_VEL
LIN {X 0,Y 376.038,Z 241.645,A -85,B 0,C 180,E1 -12251.864,E2 -12251.864} C_VEL
LIN {X 0,Y 376.047,Z 241.64,A -85,B 0,C 180,E1 -12255.168,E2 -12255.168} C_VEL
LIN {X 0,Y 376.013,Z 241.646,A -85,B 0,C 180,E1 -12258.527,E2 -12258.527} C_VEL
LIN {X 0,Y 375.954,Z 241.657,A -85,B 0,C 180,E1 -12261.955,E2 -12261.955} C_VEL
LIN {X 0,Y 375.996,Z 241.65,A -85,B 0,C 180,E1 -12265.462,E2 -12265.462} C_VEL
LIN {X 0,Y 375.967,Z 241.653,A -85,B 0,C 180,E1 -12269.079,E2 -12269.079} C_VEL
LIN {X 0,Y 375.946,Z 241.656,A -85,B 0,C 180,E1 -12272.829,E2 -12272.829} C_VEL
LIN {X 0,Y 375.948,Z 241.654,A -85,B 0,C 180,E1 -12275.417,E2 -12275.417} C_VEL
LIN {X 0,Y 375.965,Z 241.655,A -85,B 0,C 180,E1 -12278.272,E2 -12278.272} C_VEL
LIN {X 0,Y 375.924,Z 241.659,A -85,B 0,C 180,E1 -12281.602,E2 -12281.602} C_VEL
LIN {X 0,Y 375.961,Z 241.776,A -85,B 0,C 180,E1 -12284.021,E2 -12284.021} C_VEL
LIN {X 0,Y 376.742,Z 245.871,A -85,B 0,C 180,E1 -12286.68,E2 -12286.68} C_VEL
LIN {X 0,Y 377.688,Z 250.885,A -85,B 0,C 180,E1 -12289.723,E2 -12289.723} C_VEL
LIN {X 0,Y 378.585,Z 256.633,A -85,B 0,C 180,E1 -12292.963,E2 -12292.963} C_VEL
LIN {X 0,Y 378.318,Z 261.531,A -85,B 0,C 180,E1 -12295.489,E2 -12295.489} C_VEL
LIN {X 0,Y 377.515,Z 268.506,A -85,B 0,C 180,E1 -12298.91,E2 -12298.91} C_VEL
LIN {X 0,Y 376.802,Z 276.751,A -85,B 0,C 180,E1 -12302.81,E2 -12302.81} C_VEL
LIN {X 0,Y 376.033,Z 285.645,A -85,B 0,C 180,E1 -12306.893,E2 -12306.893} C_VEL
LIN {X 0,Y 375.51,Z 293.755,A -85,B 0,C 180,E1 -12310.546,E2 -12310.546} C_VEL
LIN {X 0,Y 378.038,Z 307.301,A -85,B 0,C 180,E1 -12311.134,E2 -12311.134} C_VEL
LIN {X 0,Y 379.624,Z 319.925,A -85,B 0,C 180,E1 -12311.865,E2 -12311.865} C_VEL
LIN {X 0,Y 380.532,Z 329.909,A -85,B 0,C 180,E1 -12312.584,E2 -12312.584} C_VEL
LIN {X 0,Y 379.423,Z 342.139,A -85,B 0,C 180,E1 -12313.594,E2 -12313.594} C_VEL
LIN {X 0,Y 378.342,Z 353.456,A -85,B 0,C 180,E1 -12314.79,E2 -12314.79} C_VEL
LIN {X 0,Y 377.482,Z 362.583,A -85,B 0,C 180,E1 -12315.995,E2 -12315.995} C_VEL
LIN {X 0,Y 376.708,Z 370.966,A -85,B 0,C 180,E1 -12317.339,E2 -12317.339} C_VEL
LIN {X 0,Y 375.854,Z 379.18,A -85,B 0,C 180,E1 -12318.952,E2 -12318.952} C_VEL
LIN {X 0,Y 375.395,Z 384.794,A -85,B 0,C 180,E1 -12320.301,E2 -12320.301} C_VEL
LIN {X 0,Y 374.942,Z 390.29,A -85,B 0,C 180,E1 -12321.92,E2 -12321.92} C_VEL
LIN {X 0,Y 374.698,Z 395.143,A -85,B 0,C 180,E1 -12323.77,E2 -12323.77} C_VEL
LIN {X 0,Y 374.586,Z 398.738,A -85,B 0,C 180,E1 -12325.698,E2 -12325.698} C_VEL
LIN {X 0,Y 374.59,Z 401.114,A -85,B 0,C 180,E1 -12327.851,E2 -12327.851} C_VEL
LIN {X 0,Y 374.609,Z 401.712,A -85,B 0,C 180,E1 -12328.927,E2 -12328.927} C_VEL
LIN {X 0,Y 374.604,Z 401.897,A -85,B 0,C 180,E1 -12330.002,E2 -12330.002} C_VEL
LIN {X 0,Y 374.61,Z 401.654,A -85,B 0,C 180,E1 -12331.077,E2 -12331.077} C_VEL
LIN {X 0,Y 374.622,Z 401.022,A -85,B 0,C 180,E1 -12332.152,E2 -12332.152} C_VEL
LIN {X 0,Y 374.534,Z 399.988,A -85,B 0,C 180,E1 -12333.229,E2 -12333.229} C_VEL
LIN {X 0,Y 374.588,Z 398.54,A -85,B 0,C 180,E1 -12334.306,E2 -12334.306} C_VEL
LIN {X 0,Y 374.701,Z 394.808,A -85,B 0,C 180,E1 -12336.234,E2 -12336.234} C_VEL
LIN {X 0,Y 374.952,Z 389.831,A -85,B 0,C 180,E1 -12338.083,E2 -12338.083} C_VEL
LIN {X 0,Y 375.398,Z 384.187,A -85,B 0,C 180,E1 -12339.702,E2 -12339.702} C_VEL
LIN {X 0,Y 375.963,Z 377.134,A -85,B 0,C 180,E1 -12341.321,E2 -12341.321} C_VEL
LIN {X 0,Y 376.819,Z 368.305,A -85,B 0,C 180,E1 -12342.934,E2 -12342.934} C_VEL
LIN {X 0,Y 377.739,Z 358.746,A -85,B 0,C 180,E1 -12344.346,E2 -12344.346} C_VEL
LIN {X 0,Y 378.624,Z 348.072,A -85,B 0,C 180,E1 -12345.615,E2 -12345.615} C_VEL
LIN {X 0,Y 379.588,Z 336.744,A -85,B 0,C 180,E1 -12346.679,E2 -12346.679} C_VEL
LIN {X 0,Y 380.182,Z 327.242,A -85,B 0,C 180,E1 -12347.397,E2 -12347.397} C_VEL
LIN {X 0,Y 378.711,Z 315.29,A -85,B 0,C 180,E1 -12348.186,E2 -12348.186} C_VEL
LIN {X 0,Y 376.773,Z 301.905,A -85,B 0,C 180,E1 -12348.855,E2 -12348.855} C_VEL
LIN {X 0,Y 375.472,Z 293.784,A -85,B 0,C 180,E1 -12349.183,E2 -12349.183} C_VEL
LIN {X 0,Y 375.904,Z 286.251,A -85,B 0,C 180,E1 -12352.538,E2 -12352.538} C_VEL
LIN {X 0,Y 376.567,Z 277.17,A -85,B 0,C 180,E1 -12356.612,E2 -12356.612} C_VEL
LIN {X 0,Y 377.111,Z 270.638,A -85,B 0,C 180,E1 -12359.597,E2 -12359.597} C_VEL
LIN {X 0,Y 377.846,Z 262.974,A -85,B 0,C 180,E1 -12363.174,E2 -12363.174} C_VEL
LIN {X 0,Y 378.326,Z 257.559,A -85,B 0,C 180,E1 -12365.816,E2 -12365.816} C_VEL
LIN {X 0,Y 378.104,Z 253.651,A -85,B 0,C 180,E1 -12367.836,E2 -12367.836} C_VEL
LIN {X 0,Y 377.225,Z 248.436,A -85,B 0,C 180,E1 -12370.7,E2 -12370.7} C_VEL
LIN {X 0,Y 376.058,Z 242.193,A -85,B 0,C 180,E1 -12374.37,E2 -12374.37} C_VEL
LIN {X 0,Y 375.996,Z 241.655,A -85,B 0,C 180,E1 -12374.742,E2 -12374.742} C_VEL
LIN {X 0,Y 375.941,Z 241.658,A -85,B 0,C 180,E1 -12378.4,E2 -12378.4} C_VEL
LIN {X 0,Y 375.979,Z 241.649,A -85,B 0,C 180,E1 -12381.731,E2 -12381.731} C_VEL
LIN {X 0,Y 375.985,Z 241.648,A -85,B 0,C 180,E1 -12385.334,E2 -12385.334} C_VEL
LIN {X 0,Y 375.963,Z 241.656,A -85,B 0,C 180,E1 -12388.438,E2 -12388.438} C_VEL
LIN {X 0,Y 375.965,Z 241.654,A -85,B 0,C 180,E1 -12392.139,E2 -12392.139} C_VEL
LIN {X 0,Y 375.984,Z 241.652,A -85,B 0,C 180,E1 -12394.537,E2 -12394.537} C_VEL
LIN {X 0,Y 375.967,Z 241.655,A -85,B 0,C 180,E1 -12398.046,E2 -12398.046} C_VEL
LIN {X 0,Y 376.006,Z 241.646,A -85,B 0,C 180,E1 -12401.473,E2 -12401.473} C_VEL
LIN {X 0,Y 375.997,Z 241.646,A -85,B 0,C 180,E1 -12404.83,E2 -12404.83} C_VEL
LIN {X 0,Y 376.109,Z 241.632,A -85,B 0,C 180,E1 -12407.042,E2 -12407.042} C_VEL
LIN {X 0,Y 376.116,Z 241.633,A -85,B 0,C 180,E1 -12410.319,E2 -12410.319} C_VEL
LIN {X 0,Y 376.236,Z 241.621,A -85,B 0,C 180,E1 -12413.565,E2 -12413.565} C_VEL
LIN {X 0,Y 376.359,Z 241.605,A -85,B 0,C 180,E1 -12417.86,E2 -12417.86} C_VEL
LIN {X 0,Y 376.491,Z 241.587,A -85,B 0,C 180,E1 -12420,E2 -12420} C_VEL
LIN {X 0,Y 376.351,Z 241.603,A -85,B 0,C 180,E1 -12422.141,E2 -12422.141} C_VEL
LIN {X 0,Y 376.192,Z 241.621,A -85,B 0,C 180,E1 -12426.486,E2 -12426.486} C_VEL
LIN {X 0,Y 376.118,Z 241.633,A -85,B 0,C 180,E1 -12429.682,E2 -12429.682} C_VEL
LIN {X 0,Y 376.098,Z 241.635,A -85,B 0,C 180,E1 -12433.657,E2 -12433.657} C_VEL
LIN {X 0,Y 376.041,Z 241.644,A -85,B 0,C 180,E1 -12437.4,E2 -12437.4} C_VEL
LIN {X 0,Y 375.987,Z 241.653,A -85,B 0,C 180,E1 -12440.832,E2 -12440.832} C_VEL
LIN {X 0,Y 375.942,Z 241.655,A -85,B 0,C 180,E1 -12444.285,E2 -12444.285} C_VEL
LIN {X 0,Y 375.918,Z 241.661,A -85,B 0,C 180,E1 -12446.66,E2 -12446.66} C_VEL
LIN {X 0,Y 375.921,Z 241.658,A -85,B 0,C 180,E1 -12449.084,E2 -12449.084} C_VEL
LIN {X 0,Y 375.965,Z 241.65,A -85,B 0,C 180,E1 -12451.562,E2 -12451.562} C_VEL
LIN {X 0,Y 375.965,Z 241.651,A -85,B 0,C 180,E1 -12455.415,E2 -12455.415} C_VEL
LIN {X 0,Y 375.978,Z 241.654,A -85,B 0,C 180,E1 -12458.269,E2 -12458.269} C_VEL
LIN {X 0,Y 375.94,Z 241.654,A -85,B 0,C 180,E1 -12461.6,E2 -12461.6} C_VEL
LIN {X 0,Y 375.929,Z 241.655,A -85,B 0,C 180,E1 -12465.269,E2 -12465.269} C_VEL
LIN {X 0,Y 375.919,Z 241.659,A -85,B 0,C 180,E1 -12468.402,E2 -12468.402} C_VEL
LIN {X 0,Y 375.96,Z 241.657,A -85,B 0,C 180,E1 -12471.909,E2 -12471.909} C_VEL
LIN {X 0,Y 375.981,Z 241.65,A -85,B 0,C 180,E1 -12475.333,E2 -12475.333} C_VEL
LIN {X 0,Y 375.84,Z 241.667,A -85,B 0,C 180,E1 -12478.425,E2 -12478.425} C_VEL
LIN {X 0,Y 375.531,Z 241.71,A -85,B 0,C 180,E1 -12481.594,E2 -12481.594} C_VEL
LIN {X 0,Y 375.35,Z 242.102,A -85,B 0,C 180,E1 -12483.295,E2 -12483.295} C_VEL
LIN {X 0,Y 375.262,Z 245.381,A -85,B 0,C 180,E1 -12486.839,E2 -12486.839} C_VEL
LIN {X 0,Y 375.154,Z 248.698,A -85,B 0,C 180,E1 -12490.292,E2 -12490.292} C_VEL
LIN {X 0,Y 375.134,Z 252.09,A -85,B 0,C 180,E1 -12493.677,E2 -12493.677} C_VEL
LIN {X 0,Y 375.084,Z 253.631,A -85,B 0,C 180,E1 -12495.171,E2 -12495.171} C_VEL
LIN {X 0,Y 379.02,Z 268.739,A -85,B 0,C 180,E1 -12495.966,E2 -12495.966} C_VEL
LIN {X 0,Y 380.974,Z 278.223,A -85,B 0,C 180,E1 -12496.588,E2 -12496.588} C_VEL
LIN {X 0,Y 380.498,Z 288.913,A -85,B 0,C 180,E1 -12497.328,E2 -12497.328} C_VEL
LIN {X 0,Y 379.717,Z 299.531,A -85,B 0,C 180,E1 -12498.251,E2 -12498.251} C_VEL
LIN {X 0,Y 378.986,Z 309.293,A -85,B 0,C 180,E1 -12499.312,E2 -12499.312} C_VEL
LIN {X 0,Y 378.161,Z 319.166,A -85,B 0,C 180,E1 -12500.64,E2 -12500.64} C_VEL
LIN {X 0,Y 377.366,Z 327.266,A -85,B 0,C 180,E1 -12501.969,E2 -12501.969} C_VEL
LIN {X 0,Y 376.551,Z 335.209,A -85,B 0,C 180,E1 -12503.569,E2 -12503.569} C_VEL
LIN {X 0,Y 375.871,Z 341.594,A -85,B 0,C 180,E1 -12505.172,E2 -12505.172} C_VEL
LIN {X 0,Y 375.316,Z 346.667,A -85,B 0,C 180,E1 -12506.778,E2 -12506.778} C_VEL
LIN {X 0,Y 375.03,Z 350.602,A -85,B 0,C 180,E1 -12508.388,E2 -12508.388} C_VEL
LIN {X 0,Y 374.804,Z 353.516,A -85,B 0,C 180,E1 -12509.998,E2 -12509.998} C_VEL
LIN {X 0,Y 374.755,Z 354.916,A -85,B 0,C 180,E1 -12511.073,E2 -12511.073} C_VEL
LIN {X 0,Y 374.796,Z 355.909,A -85,B 0,C 180,E1 -12512.148,E2 -12512.148} C_VEL
LIN {X 0,Y 374.791,Z 356.527,A -85,B 0,C 180,E1 -12513.223,E2 -12513.223} C_VEL
LIN {X 0,Y 374.707,Z 356.775,A -85,B 0,C 180,E1 -12514.301,E2 -12514.301} C_VEL
LIN {X 0,Y 374.809,Z 356.593,A -85,B 0,C 180,E1 -12515.378,E2 -12515.378} C_VEL
LIN {X 0,Y 374.931,Z 355.064,A -85,B 0,C 180,E1 -12517.538,E2 -12517.538} C_VEL
LIN {X 0,Y 375.029,Z 353.719,A -85,B 0,C 180,E1 -12518.621,E2 -12518.621} C_VEL
LIN {X 0,Y 375.307,Z 350.861,A -85,B 0,C 180,E1 -12520.246,E2 -12520.246} C_VEL
LIN {X 0,Y 375.745,Z 346.97,A -85,B 0,C 180,E1 -12521.871,E2 -12521.871} C_VEL
LIN {X 0,Y 376.369,Z 341.404,A -85,B 0,C 180,E1 -12523.647,E2 -12523.647} C_VEL
LIN {X 0,Y 377.204,Z 334.337,A -85,B 0,C 180,E1 -12525.395,E2 -12525.395} C_VEL
LIN {X 0,Y 378.213,Z 326.1,A -85,B 0,C 180,E1 -12527.016,E2 -12527.016} C_VEL
LIN {X 0,Y 379.148,Z 317.612,A -85,B 0,C 180,E1 -12528.366,E2 -12528.366} C_VEL
LIN {X 0,Y 380.14,Z 307.085,A -85,B 0,C 180,E1 -12529.717,E2 -12529.717} C_VEL
LIN {X 0,Y 381.175,Z 296.619,A -85,B 0,C 180,E1 -12530.787,E2 -12530.787} C_VEL
LIN {X 0,Y 382.004,Z 285.385,A -85,B 0,C 180,E1 -12531.704,E2 -12531.704} C_VEL
LIN {X 0,Y 382.095,Z 279.067,A -85,B 0,C 180,E1 -12532.139,E2 -12532.139} C_VEL
LIN {X 0,Y 378.803,Z 265.906,A -85,B 0,C 180,E1 -12533.051,E2 -12533.051} C_VEL
LIN {X 0,Y 375.17,Z 254.089,A -85,B 0,C 180,E1 -12533.71,E2 -12533.71} C_VEL
LIN {X 0,Y 371.097,Z 252.404,A -85,B 0,C 180,E1 -12535.801,E2 -12535.801} C_VEL
LIN {X 0,Y 370.028,Z 252.313,A -85,B 0,C 180,E1 -12536.418,E2 -12536.418} C_VEL
LIN {X 0,Y 368.471,Z 250.972,A -85,B 0,C 180,E1 -12537.75,E2 -12537.75} C_VEL
LIN {X 0,Y 368.297,Z 250.232,A -85,B 0,C 180,E1 -12538.428,E2 -12538.428} C_VEL
LIN {X 0,Y 368.385,Z 246.707,A -85,B 0,C 180,E1 -12542.286,E2 -12542.286} C_VEL
LIN {X 0,Y 368.541,Z 243.243,A -85,B 0,C 180,E1 -12546.237,E2 -12546.237} C_VEL
LIN {X 0,Y 368.66,Z 242.566,A -85,B 0,C 180,E1 -12547.59,E2 -12547.59} C_VEL
LIN {X 0,Y 368.847,Z 242.538,A -85,B 0,C 180,E1 -12550.376,E2 -12550.376} C_VEL
LIN {X 0,Y 368.876,Z 242.536,A -85,B 0,C 180,E1 -12553.614,E2 -12553.614} C_VEL
LIN {X 0,Y 368.878,Z 242.536,A -85,B 0,C 180,E1 -12556.694,E2 -12556.694} C_VEL
LIN {X 0,Y 368.903,Z 242.534,A -85,B 0,C 180,E1 -12559.642,E2 -12559.642} C_VEL
LIN {X 0,Y 368.894,Z 242.532,A -85,B 0,C 180,E1 -12563.143,E2 -12563.143} C_VEL
LIN {X 0,Y 368.887,Z 242.533,A -85,B 0,C 180,E1 -12566.461,E2 -12566.461} C_VEL
LIN {X 0,Y 368.92,Z 242.53,A -85,B 0,C 180,E1 -12569.045,E2 -12569.045} C_VEL
LIN {X 0,Y 368.953,Z 242.524,A -85,B 0,C 180,E1 -12572.795,E2 -12572.795} C_VEL
LIN {X 0,Y 368.935,Z 242.53,A -85,B 0,C 180,E1 -12576.112,E2 -12576.112} C_VEL
LIN {X 0,Y 368.926,Z 242.529,A -85,B 0,C 180,E1 -12579.946,E2 -12579.946} C_VEL
LIN {X 0,Y 368.965,Z 242.525,A -85,B 0,C 180,E1 -12583.398,E2 -12583.398} C_VEL
LIN {X 0,Y 369.046,Z 242.514,A -85,B 0,C 180,E1 -12586.79,E2 -12586.79} C_VEL
LIN {X 0,Y 369.055,Z 242.514,A -85,B 0,C 180,E1 -12590.131,E2 -12590.131} C_VEL
LIN {X 0,Y 369.178,Z 242.5,A -85,B 0,C 180,E1 -12592.342,E2 -12592.342} C_VEL
LIN {X 0,Y 369.141,Z 242.503,A -85,B 0,C 180,E1 -12594.537,E2 -12594.537} C_VEL
LIN {X 0,Y 369.308,Z 242.481,A -85,B 0,C 180,E1 -12597.819,E2 -12597.819} C_VEL
LIN {X 0,Y 369.444,Z 242.466,A -85,B 0,C 180,E1 -12600,E2 -12600} C_VEL
LIN {X 0,Y 369.307,Z 242.484,A -85,B 0,C 180,E1 -12602.181,E2 -12602.181} C_VEL
LIN {X 0,Y 369.204,Z 242.495,A -85,B 0,C 180,E1 -12606.558,E2 -12606.558} C_VEL
LIN {X 0,Y 369.126,Z 242.506,A -85,B 0,C 180,E1 -12608.761,E2 -12608.761} C_VEL
LIN {X 0,Y 368.993,Z 242.523,A -85,B 0,C 180,E1 -12612.094,E2 -12612.094} C_VEL
LIN {X 0,Y 368.986,Z 242.518,A -85,B 0,C 180,E1 -12615.465,E2 -12615.465} C_VEL
LIN {X 0,Y 368.972,Z 242.521,A -85,B 0,C 180,E1 -12618.893,E2 -12618.893} C_VEL
LIN {X 0,Y 368.922,Z 242.53,A -85,B 0,C 180,E1 -12622.396,E2 -12622.396} C_VEL
LIN {X 0,Y 368.989,Z 242.521,A -85,B 0,C 180,E1 -12625.981,E2 -12625.981} C_VEL
LIN {X 0,Y 368.957,Z 242.528,A -85,B 0,C 180,E1 -12628.814,E2 -12628.814} C_VEL
LIN {X 0,Y 368.9,Z 242.534,A -85,B 0,C 180,E1 -12632.238,E2 -12632.238} C_VEL
LIN {X 0,Y 368.919,Z 242.53,A -85,B 0,C 180,E1 -12635.003,E2 -12635.003} C_VEL
LIN {X 0,Y 368.899,Z 242.535,A -85,B 0,C 180,E1 -12638.641,E2 -12638.641} C_VEL
LIN {X 0,Y 368.872,Z 242.539,A -85,B 0,C 180,E1 -12642.011,E2 -12642.011} C_VEL
LIN {X 0,Y 368.91,Z 242.646,A -85,B 0,C 180,E1 -12643.525,E2 -12643.525} C_VEL
LIN {X 0,Y 369.856,Z 247.652,A -85,B 0,C 180,E1 -12646.84,E2 -12646.84} C_VEL
LIN {X 0,Y 370.786,Z 252.574,A -85,B 0,C 180,E1 -12649.878,E2 -12649.878} C_VEL
LIN {X 0,Y 371.555,Z 257.575,A -85,B 0,C 180,E1 -12652.753,E2 -12652.753} C_VEL
LIN {X 0,Y 371.499,Z 260.71,A -85,B 0,C 180,E1 -12654.437,E2 -12654.437} C_VEL
LIN {X 0,Y 370.75,Z 267.616,A -85,B 0,C 180,E1 -12657.944,E2 -12657.944} C_VEL
LIN {X 0,Y 369.833,Z 276.474,A -85,B 0,C 180,E1 -12662.254,E2 -12662.254} C_VEL
LIN {X 0,Y 369.08,Z 284.554,A -85,B 0,C 180,E1 -12666.066,E2 -12666.066} C_VEL
LIN {X 0,Y 368.638,Z 291.079,A -85,B 0,C 180,E1 -12669.096,E2 -12669.096} C_VEL
LIN {X 0,Y 368.492,Z 293.306,A -85,B 0,C 180,E1 -12670.124,E2 -12670.124} C_VEL
LIN {X 0,Y 371.1,Z 307.118,A -85,B 0,C 180,E1 -12670.749,E2 -12670.749} C_VEL
LIN {X 0,Y 372.749,Z 320.316,A -85,B 0,C 180,E1 -12671.542,E2 -12671.542} C_VEL
LIN {X 0,Y 373.712,Z 329.881,A -85,B 0,C 180,E1 -12672.26,E2 -12672.26} C_VEL
LIN {X 0,Y 372.62,Z 341.985,A -85,B 0,C 180,E1 -12673.286,E2 -12673.286} C_VEL
LIN {X 0,Y 371.465,Z 353.233,A -85,B 0,C 180,E1 -12674.502,E2 -12674.502} C_VEL
LIN {X 0,Y 370.577,Z 362.322,A -85,B 0,C 180,E1 -12675.729,E2 -12675.729} C_VEL
LIN {X 0,Y 369.766,Z 370.675,A -85,B 0,C 180,E1 -12677.097,E2 -12677.097} C_VEL
LIN {X 0,Y 368.853,Z 378.863,A -85,B 0,C 180,E1 -12678.739,E2 -12678.739} C_VEL
LIN {X 0,Y 368.343,Z 384.454,A -85,B 0,C 180,E1 -12680.114,E2 -12680.114} C_VEL
LIN {X 0,Y 367.893,Z 389.933,A -85,B 0,C 180,E1 -12681.764,E2 -12681.764} C_VEL
LIN {X 0,Y 367.643,Z 394.232,A -85,B 0,C 180,E1 -12683.415,E2 -12683.415} C_VEL
LIN {X 0,Y 367.548,Z 396.516,A -85,B 0,C 180,E1 -12684.515,E2 -12684.515} C_VEL
LIN {X 0,Y 367.516,Z 398.342,A -85,B 0,C 180,E1 -12685.615,E2 -12685.615} C_VEL
LIN {X 0,Y 367.494,Z 400.703,A -85,B 0,C 180,E1 -12687.81,E2 -12687.81} C_VEL
LIN {X 0,Y 367.544,Z 401.297,A -85,B 0,C 180,E1 -12688.906,E2 -12688.906} C_VEL
LIN {X 0,Y 367.538,Z 401.468,A -85,B 0,C 180,E1 -12690.002,E2 -12690.002} C_VEL
LIN {X 0,Y 367.546,Z 401.218,A -85,B 0,C 180,E1 -12691.097,E2 -12691.097} C_VEL
LIN {X 0,Y 367.526,Z 400.577,A -85,B 0,C 180,E1 -12692.193,E2 -12692.193} C_VEL
LIN {X 0,Y 367.447,Z 399.537,A -85,B 0,C 180,E1 -12693.291,E2 -12693.291} C_VEL
LIN {X 0,Y 367.519,Z 398.074,A -85,B 0,C 180,E1 -12694.388,E2 -12694.388} C_VEL
LIN {X 0,Y 367.601,Z 394.7,A -85,B 0,C 180,E1 -12696.191,E2 -12696.191} C_VEL
LIN {X 0,Y 367.901,Z 389.33,A -85,B 0,C 180,E1 -12698.239,E2 -12698.239} C_VEL
LIN {X 0,Y 368.345,Z 383.665,A -85,B 0,C 180,E1 -12699.889,E2 -12699.889} C_VEL
LIN {X 0,Y 368.941,Z 376.582,A -85,B 0,C 180,E1 -12701.539,E2 -12701.539} C_VEL
LIN {X 0,Y 369.837,Z 367.722,A -85,B 0,C 180,E1 -12703.183,E2 -12703.183} C_VEL
LIN {X 0,Y 370.848,Z 357.474,A -85,B 0,C 180,E1 -12704.711,E2 -12704.711} C_VEL
LIN {X 0,Y 371.725,Z 347.394,A -85,B 0,C 180,E1 -12705.913,E2 -12705.913} C_VEL
LIN {X 0,Y 372.769,Z 336.013,A -85,B 0,C 180,E1 -12706.993,E2 -12706.993} C_VEL
LIN {X 0,Y 373.252,Z 327.922,A -85,B 0,C 180,E1 -12707.625,E2 -12707.625} C_VEL
LIN {X 0,Y 371.788,Z 315.782,A -85,B 0,C 180,E1 -12708.458,E2 -12708.458} C_VEL
LIN {X 0,Y 369.861,Z 302.162,A -85,B 0,C 180,E1 -12709.166,E2 -12709.166} C_VEL
LIN {X 0,Y 368.426,Z 293.428,A -85,B 0,C 180,E1 -12709.503,E2 -12709.503} C_VEL
LIN {X 0,Y 368.89,Z 285.801,A -85,B 0,C 180,E1 -12712.991,E2 -12712.991} C_VEL
LIN {X 0,Y 369.506,Z 277.881,A -85,B 0,C 180,E1 -12716.627,E2 -12716.627} C_VEL
LIN {X 0,Y 370.183,Z 270.246,A -85,B 0,C 180,E1 -12720.207,E2 -12720.207} C_VEL
LIN {X 0,Y 370.854,Z 263.711,A -85,B 0,C 180,E1 -12723.339,E2 -12723.339} C_VEL
LIN {X 0,Y 371.318,Z 258.5,A -85,B 0,C 180,E1 -12725.928,E2 -12725.928} C_VEL
LIN {X 0,Y 371.085,Z 254.594,A -85,B 0,C 180,E1 -12727.991,E2 -12727.991} C_VEL
LIN {X 0,Y 370.286,Z 249.95,A -85,B 0,C 180,E1 -12730.606,E2 -12730.606} C_VEL
LIN {X 0,Y 369.297,Z 244.766,A -85,B 0,C 180,E1 -12733.683,E2 -12733.683} C_VEL
LIN {X 0,Y 368.938,Z 242.534,A -85,B 0,C 180,E1 -12735.185,E2 -12735.185} C_VEL
LIN {X 0,Y 368.889,Z 242.538,A -85,B 0,C 180,E1 -12738.178,E2 -12738.178} C_VEL
LIN {X 0,Y 368.913,Z 242.529,A -85,B 0,C 180,E1 -12741.361,E2 -12741.361} C_VEL
LIN {X 0,Y 368.942,Z 242.526,A -85,B 0,C 180,E1 -12745.147,E2 -12745.147} C_VEL
LIN {X 0,Y 368.92,Z 242.529,A -85,B 0,C 180,E1 -12749.046,E2 -12749.046} C_VEL
LIN {X 0,Y 368.938,Z 242.526,A -85,B 0,C 180,E1 -12751.56,E2 -12751.56} C_VEL
LIN {X 0,Y 368.947,Z 242.524,A -85,B 0,C 180,E1 -12755.224,E2 -12755.224} C_VEL
LIN {X 0,Y 368.927,Z 242.527,A -85,B 0,C 180,E1 -12758.981,E2 -12758.981} C_VEL
LIN {X 0,Y 368.98,Z 242.524,A -85,B 0,C 180,E1 -12762.257,E2 -12762.257} C_VEL
LIN {X 0,Y 369.045,Z 242.515,A -85,B 0,C 180,E1 -12766.228,E2 -12766.228} C_VEL
LIN {X 0,Y 369.066,Z 242.513,A -85,B 0,C 180,E1 -12770.132,E2 -12770.132} C_VEL
LIN {X 0,Y 369.195,Z 242.497,A -85,B 0,C 180,E1 -12773.442,E2 -12773.442} C_VEL
LIN {X 0,Y 369.324,Z 242.481,A -85,B 0,C 180,E1 -12777.819,E2 -12777.819} C_VEL
LIN {X 0,Y 369.461,Z 242.462,A -85,B 0,C 180,E1 -12780,E2 -12780} C_VEL
LIN {X 0,Y 369.315,Z 242.479,A -85,B 0,C 180,E1 -12782.181,E2 -12782.181} C_VEL
LIN {X 0,Y 369.159,Z 242.498,A -85,B 0,C 180,E1 -12786.559,E2 -12786.559} C_VEL
LIN {X 0,Y 369.069,Z 242.51,A -85,B 0,C 180,E1 -12789.868,E2 -12789.868} C_VEL
LIN {X 0,Y 369.046,Z 242.513,A -85,B 0,C 180,E1 -12793.772,E2 -12793.772} C_VEL
LIN {X 0,Y 368.999,Z 242.518,A -85,B 0,C 180,E1 -12797.743,E2 -12797.743} C_VEL
LIN {X 0,Y 368.917,Z 242.531,A -85,B 0,C 180,E1 -12801.221,E2 -12801.221} C_VEL
LIN {X 0,Y 368.915,Z 242.528,A -85,B 0,C 180,E1 -12803.873,E2 -12803.873} C_VEL
LIN {X 0,Y 368.864,Z 242.536,A -85,B 0,C 180,E1 -12807.212,E2 -12807.212} C_VEL
LIN {X 0,Y 368.9,Z 242.53,A -85,B 0,C 180,E1 -12809.692,E2 -12809.692} C_VEL
LIN {X 0,Y 368.905,Z 242.531,A -85,B 0,C 180,E1 -12813.043,E2 -12813.043} C_VEL
LIN {X 0,Y 368.924,Z 242.531,A -85,B 0,C 180,E1 -12816.196,E2 -12816.196} C_VEL
LIN {X 0,Y 368.906,Z 242.531,A -85,B 0,C 180,E1 -12818.953,E2 -12818.953} C_VEL
LIN {X 0,Y 368.888,Z 242.535,A -85,B 0,C 180,E1 -12822.009,E2 -12822.009} C_VEL
LIN {X 0,Y 368.882,Z 242.532,A -85,B 0,C 180,E1 -12825.174,E2 -12825.174} C_VEL
LIN {X 0,Y 368.867,Z 242.539,A -85,B 0,C 180,E1 -12828.174,E2 -12828.174} C_VEL
LIN {X 0,Y 368.883,Z 242.533,A -85,B 0,C 180,E1 -12831.365,E2 -12831.365} C_VEL
LIN {X 0,Y 368.937,Z 242.526,A -85,B 0,C 180,E1 -12835.145,E2 -12835.145} C_VEL
LIN {X 0,Y 368.838,Z 242.544,A -85,B 0,C 180,E1 -12837.755,E2 -12837.755} C_VEL
LIN {X 0,Y 368.529,Z 242.579,A -85,B 0,C 180,E1 -12841.312,E2 -12841.312} C_VEL
LIN {X 0,Y 368.337,Z 242.607,A -85,B 0,C 180,E1 -12842.745,E2 -12842.745} C_VEL
LIN {X 0,Y 368.232,Z 244.675,A -85,B 0,C 180,E1 -12845.171,E2 -12845.171} C_VEL
LIN {X 0,Y 368.123,Z 248.011,A -85,B 0,C 180,E1 -12848.73,E2 -12848.73} C_VEL
LIN {X 0,Y 368.079,Z 251.857,A -85,B 0,C 180,E1 -12852.687,E2 -12852.687} C_VEL
LIN {X 0,Y 368.042,Z 254.093,A -85,B 0,C 180,E1 -12854.854,E2 -12854.854} C_VEL
LIN {X 0,Y 371.533,Z 267.281,A -85,B 0,C 180,E1 -12855.531,E2 -12855.531} C_VEL
LIN {X 0,Y 374.156,Z 279.422,A -85,B 0,C 180,E1 -12856.336,E2 -12856.336} C_VEL
LIN {X 0,Y 373.524,Z 291.614,A -85,B 0,C 180,E1 -12857.226,E2 -12857.226} C_VEL
LIN {X 0,Y 372.648,Z 303.017,A -85,B 0,C 180,E1 -12858.301,E2 -12858.301} C_VEL
LIN {X 0,Y 371.805,Z 313.017,A -85,B 0,C 180,E1 -12859.481,E2 -12859.481} C_VEL
LIN {X 0,Y 371.002,Z 321.68,A -85,B 0,C 180,E1 -12860.732,E2 -12860.732} C_VEL
LIN {X 0,Y 370.245,Z 329.427,A -85,B 0,C 180,E1 -12862.088,E2 -12862.088} C_VEL
LIN {X 0,Y 369.419,Z 337.003,A -85,B 0,C 180,E1 -12863.718,E2 -12863.718} C_VEL
LIN {X 0,Y 368.825,Z 342.195,A -85,B 0,C 180,E1 -12865.079,E2 -12865.079} C_VEL
LIN {X 0,Y 368.255,Z 347.227,A -85,B 0,C 180,E1 -12866.716,E2 -12866.716} C_VEL
LIN {X 0,Y 367.976,Z 351.129,A -85,B 0,C 180,E1 -12868.357,E2 -12868.357} C_VEL
LIN {X 0,Y 367.727,Z 354.019,A -85,B 0,C 180,E1 -12869.998,E2 -12869.998} C_VEL
LIN {X 0,Y 367.731,Z 356.371,A -85,B 0,C 180,E1 -12872.189,E2 -12872.189} C_VEL
LIN {X 0,Y 367.695,Z 356.977,A -85,B 0,C 180,E1 -12873.286,E2 -12873.286} C_VEL
LIN {X 0,Y 367.636,Z 357.204,A -85,B 0,C 180,E1 -12874.384,E2 -12874.384} C_VEL
LIN {X 0,Y 367.778,Z 356.513,A -85,B 0,C 180,E1 -12876.438,E2 -12876.438} C_VEL
LIN {X 0,Y 367.864,Z 355.441,A -85,B 0,C 180,E1 -12877.684,E2 -12877.684} C_VEL
LIN {X 0,Y 367.978,Z 354.075,A -85,B 0,C 180,E1 -12878.787,E2 -12878.787} C_VEL
LIN {X 0,Y 368.279,Z 351.191,A -85,B 0,C 180,E1 -12880.443,E2 -12880.443} C_VEL
LIN {X 0,Y 368.769,Z 347.267,A -85,B 0,C 180,E1 -12882.099,E2 -12882.099} C_VEL
LIN {X 0,Y 369.487,Z 341.128,A -85,B 0,C 180,E1 -12884.052,E2 -12884.052} C_VEL
LIN {X 0,Y 370.317,Z 334.539,A -85,B 0,C 180,E1 -12885.689,E2 -12885.689} C_VEL
LIN {X 0,Y 371.377,Z 326.251,A -85,B 0,C 180,E1 -12887.339,E2 -12887.339} C_VEL
LIN {X 0,Y 372.515,Z 316.36,A -85,B 0,C 180,E1 -12888.899,E2 -12888.899} C_VEL
LIN {X 0,Y 373.56,Z 305.906,A -85,B 0,C 180,E1 -12890.223,E2 -12890.223} C_VEL
LIN {X 0,Y 374.671,Z 295.016,A -85,B 0,C 180,E1 -12891.309,E2 -12891.309} C_VEL
LIN {X 0,Y 375.491,Z 282.813,A -85,B 0,C 180,E1 -12892.266,E2 -12892.266} C_VEL
LIN {X 0,Y 375.253,Z 280.031,A -85,B 0,C 180,E1 -12892.476,E2 -12892.476} C_VEL
LIN {X 0,Y 372.063,Z 267.337,A -85,B 0,C 180,E1 -12893.391,E2 -12893.391} C_VEL
LIN {X 0,Y 368.129,Z 254.337,A -85,B 0,C 180,E1 -12894.137,E2 -12894.137} C_VEL
LIN {X 0,Y 368.218,Z 251.315,A -85,B 0,C 180,E1 -12897.261,E2 -12897.261} C_VEL
LIN {X 0,Y 368.297,Z 250.232,A -85,B 0,C 180,E1 -12898.428,E2 -12898.428} C_VEL
LIN {X 0,Y 367.724,Z 249.479,A -85,B 0,C 180,E1 -12899.333,E2 -12899.333} C_VEL
LIN {X 0,Y 364.918,Z 248.501,A -85,B 0,C 180,E1 -12900.812,E2 -12900.812} C_VEL
LIN {X 0,Y 362.497,Z 247.746,A -85,B 0,C 180,E1 -12902.009,E2 -12902.009} C_VEL
LIN {X 0,Y 361.466,Z 247.064,A -85,B 0,C 180,E1 -12902.933,E2 -12902.933} C_VEL
LIN {X 0,Y 361.39,Z 246.798,A -85,B 0,C 180,E1 -12903.245,E2 -12903.245} C_VEL
LIN {X 0,Y 361.552,Z 243.459,A -85,B 0,C 180,E1 -12907.157,E2 -12907.157} C_VEL
LIN {X 0,Y 361.755,Z 243.423,A -85,B 0,C 180,E1 -12909.872,E2 -12909.872} C_VEL
LIN {X 0,Y 361.827,Z 243.417,A -85,B 0,C 180,E1 -12912.828,E2 -12912.828} C_VEL
LIN {X 0,Y 361.811,Z 243.418,A -85,B 0,C 180,E1 -12915.945,E2 -12915.945} C_VEL
LIN {X 0,Y 361.827,Z 243.415,A -85,B 0,C 180,E1 -12919.243,E2 -12919.243} C_VEL
LIN {X 0,Y 361.862,Z 243.41,A -85,B 0,C 180,E1 -12922.774,E2 -12922.774} C_VEL
LIN {X 0,Y 361.846,Z 243.412,A -85,B 0,C 180,E1 -12925.718,E2 -12925.718} C_VEL
LIN {X 0,Y 361.863,Z 243.409,A -85,B 0,C 180,E1 -12929.671,E2 -12929.671} C_VEL
LIN {X 0,Y 361.944,Z 243.397,A -85,B 0,C 180,E1 -12933.474,E2 -12933.474} C_VEL
LIN {X 0,Y 361.88,Z 243.409,A -85,B 0,C 180,E1 -12937.144,E2 -12937.144} C_VEL
LIN {X 0,Y 361.896,Z 243.408,A -85,B 0,C 180,E1 -12940.723,E2 -12940.723} C_VEL
LIN {X 0,Y 361.922,Z 243.402,A -85,B 0,C 180,E1 -12943.065,E2 -12943.065} C_VEL
LIN {X 0,Y 361.987,Z 243.392,A -85,B 0,C 180,E1 -12946.527,E2 -12946.527} C_VEL
LIN {X 0,Y 362.019,Z 243.39,A -85,B 0,C 180,E1 -12949.937,E2 -12949.937} C_VEL
LIN {X 0,Y 362.136,Z 243.379,A -85,B 0,C 180,E1 -12952.192,E2 -12952.192} C_VEL
LIN {X 0,Y 362.114,Z 243.379,A -85,B 0,C 180,E1 -12954.431,E2 -12954.431} C_VEL
LIN {X 0,Y 362.273,Z 243.358,A -85,B 0,C 180,E1 -12957.776,E2 -12957.776} C_VEL
LIN {X 0,Y 362.413,Z 243.341,A -85,B 0,C 180,E1 -12960,E2 -12960} C_VEL
LIN {X 0,Y 362.271,Z 243.36,A -85,B 0,C 180,E1 -12962.223,E2 -12962.223} C_VEL
LIN {X 0,Y 362.166,Z 243.372,A -85,B 0,C 180,E1 -12966.686,E2 -12966.686} C_VEL
LIN {X 0,Y 362.062,Z 243.386,A -85,B 0,C 180,E1 -12968.933,E2 -12968.933} C_VEL
LIN {X 0,Y 361.948,Z 243.398,A -85,B 0,C 180,E1 -12972.333,E2 -12972.333} C_VEL
LIN {X 0,Y 361.95,Z 243.397,A -85,B 0,C 180,E1 -12974.621,E2 -12974.621} C_VEL
LIN {X 0,Y 361.948,Z 243.399,A -85,B 0,C 180,E1 -12978.1,E2 -12978.1} C_VEL
LIN {X 0,Y 361.881,Z 243.409,A -85,B 0,C 180,E1 -12981.654,E2 -12981.654} C_VEL
LIN {X 0,Y 361.918,Z 243.405,A -85,B 0,C 180,E1 -12985.291,E2 -12985.291} C_VEL
LIN {X 0,Y 361.912,Z 243.403,A -85,B 0,C 180,E1 -12987.779,E2 -12987.779} C_VEL
LIN {X 0,Y 361.849,Z 243.413,A -85,B 0,C 180,E1 -12991.628,E2 -12991.628} C_VEL
LIN {X 0,Y 361.865,Z 243.408,A -85,B 0,C 180,E1 -12995.346,E2 -12995.346} C_VEL
LIN {X 0,Y 361.86,Z 243.41,A -85,B 0,C 180,E1 -12999.028,E2 -12999.028} C_VEL
LIN {X 0,Y 361.855,Z 243.534,A -85,B 0,C 180,E1 -13003.016,E2 -13003.016} C_VEL
LIN {X 0,Y 362.855,Z 248.737,A -85,B 0,C 180,E1 -13006.579,E2 -13006.579} C_VEL
LIN {X 0,Y 363.778,Z 253.665,A -85,B 0,C 180,E1 -13009.685,E2 -13009.685} C_VEL
LIN {X 0,Y 364.467,Z 257.986,A -85,B 0,C 180,E1 -13012.242,E2 -13012.242} C_VEL
LIN {X 0,Y 364.543,Z 261.269,A -85,B 0,C 180,E1 -13014.068,E2 -13014.068} C_VEL
LIN {X 0,Y 363.862,Z 267.379,A -85,B 0,C 180,E1 -13017.263,E2 -13017.263} C_VEL
LIN {X 0,Y 363.018,Z 274.939,A -85,B 0,C 180,E1 -13021.055,E2 -13021.055} C_VEL
LIN {X 0,Y 362.378,Z 281.227,A -85,B 0,C 180,E1 -13024.13,E2 -13024.13} C_VEL
LIN {X 0,Y 361.76,Z 288.776,A -85,B 0,C 180,E1 -13027.741,E2 -13027.741} C_VEL
LIN {X 0,Y 361.488,Z 293.007,A -85,B 0,C 180,E1 -13029.697,E2 -13029.697} C_VEL
LIN {X 0,Y 364.129,Z 306.509,A -85,B 0,C 180,E1 -13030.326,E2 -13030.326} C_VEL
LIN {X 0,Y 365.699,Z 318.494,A -85,B 0,C 180,E1 -13031.053,E2 -13031.053} C_VEL
LIN {X 0,Y 366.842,Z 331.285,A -85,B 0,C 180,E1 -13032.037,E2 -13032.037} C_VEL
LIN {X 0,Y 365.667,Z 343.249,A -85,B 0,C 180,E1 -13033.102,E2 -13033.102} C_VEL
LIN {X 0,Y 364.481,Z 354.09,A -85,B 0,C 180,E1 -13034.34,E2 -13034.34} C_VEL
LIN {X 0,Y 363.459,Z 363.858,A -85,B 0,C 180,E1 -13035.729,E2 -13035.729} C_VEL
LIN {X 0,Y 362.628,Z 371.885,A -85,B 0,C 180,E1 -13037.124,E2 -13037.124} C_VEL
LIN {X 0,Y 361.708,Z 379.77,A -85,B 0,C 180,E1 -13038.798,E2 -13038.798} C_VEL
LIN {X 0,Y 361.128,Z 386.091,A -85,B 0,C 180,E1 -13040.48,E2 -13040.48} C_VEL
LIN {X 0,Y 360.717,Z 391.137,A -85,B 0,C 180,E1 -13042.163,E2 -13042.163} C_VEL
LIN {X 0,Y 360.512,Z 395.036,A -85,B 0,C 180,E1 -13043.837,E2 -13043.837} C_VEL
LIN {X 0,Y 360.446,Z 397.948,A -85,B 0,C 180,E1 -13045.529,E2 -13045.529} C_VEL
LIN {X 0,Y 360.398,Z 400.294,A -85,B 0,C 180,E1 -13047.766,E2 -13047.766} C_VEL
LIN {X 0,Y 360.48,Z 400.882,A -85,B 0,C 180,E1 -13048.885,E2 -13048.885} C_VEL
LIN {X 0,Y 360.473,Z 401.038,A -85,B 0,C 180,E1 -13050.002,E2 -13050.002} C_VEL
LIN {X 0,Y 360.483,Z 400.782,A -85,B 0,C 180,E1 -13051.119,E2 -13051.119} C_VEL
LIN {X 0,Y 360.43,Z 400.13,A -85,B 0,C 180,E1 -13052.237,E2 -13052.237} C_VEL
LIN {X 0,Y 360.364,Z 399.083,A -85,B 0,C 180,E1 -13053.356,E2 -13053.356} C_VEL
LIN {X 0,Y 360.45,Z 397.606,A -85,B 0,C 180,E1 -13054.475,E2 -13054.475} C_VEL
LIN {X 0,Y 360.528,Z 394.5,A -85,B 0,C 180,E1 -13056.186,E2 -13056.186} C_VEL
LIN {X 0,Y 360.723,Z 390.461,A -85,B 0,C 180,E1 -13057.84,E2 -13057.84} C_VEL
LIN {X 0,Y 361.226,Z 384.161,A -85,B 0,C 180,E1 -13059.803,E2 -13059.803} C_VEL
LIN {X 0,Y 361.834,Z 377.302,A -85,B 0,C 180,E1 -13061.485,E2 -13061.485} C_VEL
LIN {X 0,Y 362.744,Z 368.781,A -85,B 0,C 180,E1 -13063.16,E2 -13063.16} C_VEL
LIN {X 0,Y 363.743,Z 358.904,A -85,B 0,C 180,E1 -13064.708,E2 -13064.708} C_VEL
LIN {X 0,Y 364.732,Z 347.995,A -85,B 0,C 180,E1 -13066.082,E2 -13066.082} C_VEL
LIN {X 0,Y 365.788,Z 336.858,A -85,B 0,C 180,E1 -13067.183,E2 -13067.183} C_VEL
LIN {X 0,Y 366.361,Z 330.145,A -85,B 0,C 180,E1 -13067.732,E2 -13067.732} C_VEL
LIN {X 0,Y 365.01,Z 317.278,A -85,B 0,C 180,E1 -13068.678,E2 -13068.678} C_VEL
LIN {X 0,Y 363.202,Z 304.083,A -85,B 0,C 180,E1 -13069.408,E2 -13069.408} C_VEL
LIN {X 0,Y 361.384,Z 293.054,A -85,B 0,C 180,E1 -13069.861,E2 -13069.861} C_VEL
LIN {X 0,Y 361.864,Z 285.347,A -85,B 0,C 180,E1 -13073.464,E2 -13073.464} C_VEL
LIN {X 0,Y 362.473,Z 278.07,A -85,B 0,C 180,E1 -13076.887,E2 -13076.887} C_VEL
LIN {X 0,Y 363.126,Z 271.139,A -85,B 0,C 180,E1 -13080.214,E2 -13080.214} C_VEL
LIN {X 0,Y 363.812,Z 264.834,A -85,B 0,C 180,E1 -13083.309,E2 -13083.309} C_VEL
LIN {X 0,Y 364.299,Z 259.775,A -85,B 0,C 180,E1 -13085.879,E2 -13085.879} C_VEL
LIN {X 0,Y 364.055,Z 255.555,A -85,B 0,C 180,E1 -13088.154,E2 -13088.154} C_VEL
LIN {X 0,Y 362.95,Z 249.166,A -85,B 0,C 180,E1 -13091.859,E2 -13091.859} C_VEL
LIN {X 0,Y 361.893,Z 243.412,A -85,B 0,C 180,E1 -13095.497,E2 -13095.497} C_VEL
LIN {X 0,Y 361.842,Z 243.415,A -85,B 0,C 180,E1 -13099.246,E2 -13099.246} C_VEL
LIN {X 0,Y 361.869,Z 243.41,A -85,B 0,C 180,E1 -13102.778,E2 -13102.778} C_VEL
LIN {X 0,Y 361.86,Z 243.407,A -85,B 0,C 180,E1 -13105.72,E2 -13105.72} C_VEL
LIN {X 0,Y 361.865,Z 243.407,A -85,B 0,C 180,E1 -13109.671,E2 -13109.671} C_VEL
LIN {X 0,Y 361.908,Z 243.401,A -85,B 0,C 180,E1 -13113.471,E2 -13113.471} C_VEL
LIN {X 0,Y 361.89,Z 243.403,A -85,B 0,C 180,E1 -13117.145,E2 -13117.145} C_VEL
LIN {X 0,Y 361.882,Z 243.405,A -85,B 0,C 180,E1 -13120.722,E2 -13120.722} C_VEL
LIN {X 0,Y 361.903,Z 243.405,A -85,B 0,C 180,E1 -13124.224,E2 -13124.224} C_VEL
LIN {X 0,Y 362.006,Z 243.39,A -85,B 0,C 180,E1 -13126.528,E2 -13126.528} C_VEL
LIN {X 0,Y 362.003,Z 243.394,A -85,B 0,C 180,E1 -13129.937,E2 -13129.937} C_VEL
LIN {X 0,Y 362.155,Z 243.372,A -85,B 0,C 180,E1 -13133.314,E2 -13133.314} C_VEL
LIN {X 0,Y 362.288,Z 243.358,A -85,B 0,C 180,E1 -13137.777,E2 -13137.777} C_VEL
LIN {X 0,Y 362.41,Z 243.34,A -85,B 0,C 180,E1 -13140,E2 -13140} C_VEL
LIN {X 0,Y 362.278,Z 243.355,A -85,B 0,C 180,E1 -13142.224,E2 -13142.224} C_VEL
LIN {X 0,Y 362.124,Z 243.375,A -85,B 0,C 180,E1 -13146.687,E2 -13146.687} C_VEL
LIN {X 0,Y 362.006,Z 243.389,A -85,B 0,C 180,E1 -13150.063,E2 -13150.063} C_VEL
LIN {X 0,Y 362.006,Z 243.389,A -85,B 0,C 180,E1 -13153.899,E2 -13153.899} C_VEL
LIN {X 0,Y 361.936,Z 243.403,A -85,B 0,C 180,E1 -13156.934,E2 -13156.934} C_VEL
LIN {X 0,Y 361.895,Z 243.405,A -85,B 0,C 180,E1 -13160.461,E2 -13160.461} C_VEL
LIN {X 0,Y 361.869,Z 243.406,A -85,B 0,C 180,E1 -13164.101,E2 -13164.101} C_VEL
LIN {X 0,Y 361.842,Z 243.409,A -85,B 0,C 180,E1 -13167.785,E2 -13167.785} C_VEL
LIN {X 0,Y 361.855,Z 243.408,A -85,B 0,C 180,E1 -13171.285,E2 -13171.285} C_VEL
LIN {X 0,Y 361.862,Z 243.411,A -85,B 0,C 180,E1 -13174.28,E2 -13174.28} C_VEL
LIN {X 0,Y 361.87,Z 243.406,A -85,B 0,C 180,E1 -13177.222,E2 -13177.222} C_VEL
LIN {X 0,Y 361.841,Z 243.411,A -85,B 0,C 180,E1 -13180.754,E2 -13180.754} C_VEL
LIN {X 0,Y 361.822,Z 243.416,A -85,B 0,C 180,E1 -13184.368,E2 -13184.368} C_VEL
LIN {X 0,Y 361.829,Z 243.412,A -85,B 0,C 180,E1 -13187.57,E2 -13187.57} C_VEL
LIN {X 0,Y 361.85,Z 243.41,A -85,B 0,C 180,E1 -13191.571,E2 -13191.571} C_VEL
LIN {X 0,Y 361.877,Z 243.405,A -85,B 0,C 180,E1 -13194.655,E2 -13194.655} C_VEL
LIN {X 0,Y 361.825,Z 243.412,A -85,B 0,C 180,E1 -13197.051,E2 -13197.051} C_VEL
LIN {X 0,Y 361.637,Z 243.44,A -85,B 0,C 180,E1 -13199.648,E2 -13199.648} C_VEL
LIN {X 0,Y 361.362,Z 243.474,A -85,B 0,C 180,E1 -13202.174,E2 -13202.174} C_VEL
LIN {X 0,Y 361.267,Z 244.026,A -85,B 0,C 180,E1 -13203.493,E2 -13203.493} C_VEL
LIN {X 0,Y 361.116,Z 247.311,A -85,B 0,C 180,E1 -13207.091,E2 -13207.091} C_VEL
LIN {X 0,Y 361.021,Z 250.689,A -85,B 0,C 180,E1 -13210.673,E2 -13210.673} C_VEL
LIN {X 0,Y 361.036,Z 252.991,A -85,B 0,C 180,E1 -13213.021,E2 -13213.021} C_VEL
LIN {X 0,Y 360.985,Z 254.444,A -85,B 0,C 180,E1 -13214.471,E2 -13214.471} C_VEL
LIN {X 0,Y 365.066,Z 269.943,A -85,B 0,C 180,E1 -13215.326,E2 -13215.326} C_VEL
LIN {X 0,Y 367.293,Z 280.553,A -85,B 0,C 180,E1 -13216.069,E2 -13216.069} C_VEL
LIN {X 0,Y 366.667,Z 292.61,A -85,B 0,C 180,E1 -13216.983,E2 -13216.983} C_VEL
LIN {X 0,Y 365.767,Z 303.907,A -85,B 0,C 180,E1 -13218.078,E2 -13218.078} C_VEL
LIN {X 0,Y 364.861,Z 314.062,A -85,B 0,C 180,E1 -13219.31,E2 -13219.31} C_VEL
LIN {X 0,Y 364.031,Z 322.426,A -85,B 0,C 180,E1 -13220.553,E2 -13220.553} C_VEL
LIN {X 0,Y 363.268,Z 330.111,A -85,B 0,C 180,E1 -13221.935,E2 -13221.935} C_VEL
LIN {X 0,Y 362.401,Z 337.631,A -85,B 0,C 180,E1 -13223.596,E2 -13223.596} C_VEL
LIN {X 0,Y 361.783,Z 342.788,A -85,B 0,C 180,E1 -13224.983,E2 -13224.983} C_VEL
LIN {X 0,Y 361.197,Z 347.782,A -85,B 0,C 180,E1 -13226.652,E2 -13226.652} C_VEL
LIN {X 0,Y 360.923,Z 351.651,A -85,B 0,C 180,E1 -13228.325,E2 -13228.325} C_VEL
LIN {X 0,Y 360.653,Z 354.517,A -85,B 0,C 180,E1 -13229.998,E2 -13229.998} C_VEL
LIN {X 0,Y 360.666,Z 356.833,A -85,B 0,C 180,E1 -13232.232,E2 -13232.232} C_VEL
LIN {X 0,Y 360.601,Z 357.426,A -85,B 0,C 180,E1 -13233.35,E2 -13233.35} C_VEL
LIN {X 0,Y 360.566,Z 357.629,A -85,B 0,C 180,E1 -13234.47,E2 -13234.47} C_VEL
LIN {X 0,Y 360.709,Z 356.989,A -85,B 0,C 180,E1 -13236.443,E2 -13236.443} C_VEL
LIN {X 0,Y 360.803,Z 355.818,A -85,B 0,C 180,E1 -13237.835,E2 -13237.835} C_VEL
LIN {X 0,Y 360.943,Z 354.427,A -85,B 0,C 180,E1 -13238.96,E2 -13238.96} C_VEL
LIN {X 0,Y 361.264,Z 351.517,A -85,B 0,C 180,E1 -13240.648,E2 -13240.648} C_VEL
LIN {X 0,Y 361.798,Z 347.559,A -85,B 0,C 180,E1 -13242.336,E2 -13242.336} C_VEL
LIN {X 0,Y 362.526,Z 341.713,A -85,B 0,C 180,E1 -13244.23,E2 -13244.23} C_VEL
LIN {X 0,Y 363.431,Z 334.743,A -85,B 0,C 180,E1 -13245.994,E2 -13245.994} C_VEL
LIN {X 0,Y 364.556,Z 326.394,A -85,B 0,C 180,E1 -13247.674,E2 -13247.674} C_VEL
LIN {X 0,Y 365.74,Z 316.603,A -85,B 0,C 180,E1 -13249.237,E2 -13249.237} C_VEL
LIN {X 0,Y 366.714,Z 307.081,A -85,B 0,C 180,E1 -13250.471,E2 -13250.471} C_VEL
LIN {X 0,Y 367.872,Z 296.426,A -85,B 0,C 180,E1 -13251.576,E2 -13251.576} C_VEL
LIN {X 0,Y 368.811,Z 283.903,A -85,B 0,C 180,E1 -13252.589,E2 -13252.589} C_VEL
LIN {X 0,Y 367.463,Z 276.848,A -85,B 0,C 180,E1 -13253.157,E2 -13253.157} C_VEL
LIN {X 0,Y 364.188,Z 264.751,A -85,B 0,C 180,E1 -13254.009,E2 -13254.009} C_VEL
LIN {X 0,Y 361.096,Z 254.757,A -85,B 0,C 180,E1 -13254.591,E2 -13254.591} C_VEL
LIN {X 0,Y 361.216,Z 251.666,A -85,B 0,C 180,E1 -13257.835,E2 -13257.835} C_VEL
LIN {X 0,Y 361.314,Z 248.192,A -85,B 0,C 180,E1 -13261.678,E2 -13261.678} C_VEL
LIN {X 0,Y 361.39,Z 246.798,A -85,B 0,C 180,E1 -13263.245,E2 -13263.245} C_VEL
LIN {X 0,Y 360.76,Z 246.08,A -85,B 0,C 180,E1 -13264.169,E2 -13264.169} C_VEL
LIN {X 0,Y 357.992,Z 245.192,A -85,B 0,C 180,E1 -13265.679,E2 -13265.679} C_VEL
LIN {X 0,Y 355.646,Z 244.596,A -85,B 0,C 180,E1 -13266.904,E2 -13266.904} C_VEL
LIN {X 0,Y 354.653,Z 244.339,A -85,B 0,C 180,E1 -13267.852,E2 -13267.852} C_VEL
LIN {X 0,Y 354.58,Z 244.316,A -85,B 0,C 180,E1 -13268.172,E2 -13268.172} C_VEL
LIN {X 0,Y 354.752,Z 244.296,A -85,B 0,C 180,E1 -13271.164,E2 -13271.164} C_VEL
LIN {X 0,Y 354.757,Z 244.297,A -85,B 0,C 180,E1 -13274.505,E2 -13274.505} C_VEL
LIN {X 0,Y 354.786,Z 244.293,A -85,B 0,C 180,E1 -13277.661,E2 -13277.661} C_VEL
LIN {X 0,Y 354.807,Z 244.291,A -85,B 0,C 180,E1 -13280.665,E2 -13280.665} C_VEL
LIN {X 0,Y 354.814,Z 244.29,A -85,B 0,C 180,E1 -13284.299,E2 -13284.299} C_VEL
LIN {X 0,Y 354.778,Z 244.294,A -85,B 0,C 180,E1 -13287.665,E2 -13287.665} C_VEL
LIN {X 0,Y 354.837,Z 244.283,A -85,B 0,C 180,E1 -13291.617,E2 -13291.617} C_VEL
LIN {X 0,Y 354.889,Z 244.281,A -85,B 0,C 180,E1 -13294.172,E2 -13294.172} C_VEL
LIN {X 0,Y 354.824,Z 244.287,A -85,B 0,C 180,E1 -13297.893,E2 -13297.893} C_VEL
LIN {X 0,Y 354.911,Z 244.275,A -85,B 0,C 180,E1 -13301.891,E2 -13301.891} C_VEL
LIN {X 0,Y 354.931,Z 244.273,A -85,B 0,C 180,E1 -13305.98,E2 -13305.98} C_VEL
LIN {X 0,Y 354.966,Z 244.268,A -85,B 0,C 180,E1 -13309.735,E2 -13309.735} C_VEL
LIN {X 0,Y 355.117,Z 244.252,A -85,B 0,C 180,E1 -13312.037,E2 -13312.037} C_VEL
LIN {X 0,Y 355.088,Z 244.255,A -85,B 0,C 180,E1 -13314.32,E2 -13314.32} C_VEL
LIN {X 0,Y 355.236,Z 244.234,A -85,B 0,C 180,E1 -13317.732,E2 -13317.732} C_VEL
LIN {X 0,Y 355.362,Z 244.22,A -85,B 0,C 180,E1 -13320,E2 -13320} C_VEL
LIN {X 0,Y 355.235,Z 244.237,A -85,B 0,C 180,E1 -13322.268,E2 -13322.268} C_VEL
LIN {X 0,Y 355.131,Z 244.249,A -85,B 0,C 180,E1 -13326.819,E2 -13326.819} C_VEL
LIN {X 0,Y 355.003,Z 244.265,A -85,B 0,C 180,E1 -13329.113,E2 -13329.113} C_VEL
LIN {X 0,Y 354.909,Z 244.274,A -85,B 0,C 180,E1 -13332.581,E2 -13332.581} C_VEL
LIN {X 0,Y 354.878,Z 244.276,A -85,B 0,C 180,E1 -13336.096,E2 -13336.096} C_VEL
LIN {X 0,Y 354.895,Z 244.276,A -85,B 0,C 180,E1 -13338.472,E2 -13338.472} C_VEL
LIN {X 0,Y 354.824,Z 244.288,A -85,B 0,C 180,E1 -13342.107,E2 -13342.107} C_VEL
LIN {X 0,Y 354.889,Z 244.278,A -85,B 0,C 180,E1 -13345.828,E2 -13345.828} C_VEL
LIN {X 0,Y 354.844,Z 244.285,A -85,B 0,C 180,E1 -13349.679,E2 -13349.679} C_VEL
LIN {X 0,Y 354.821,Z 244.288,A -85,B 0,C 180,E1 -13353.683,E2 -13353.683} C_VEL
LIN {X 0,Y 354.789,Z 244.293,A -85,B 0,C 180,E1 -13356.461,E2 -13356.461} C_VEL
LIN {X 0,Y 354.815,Z 244.286,A -85,B 0,C 180,E1 -13359.425,E2 -13359.425} C_VEL
LIN {X 0,Y 354.793,Z 244.373,A -85,B 0,C 180,E1 -13362.478,E2 -13362.478} C_VEL
LIN {X 0,Y 355.82,Z 249.772,A -85,B 0,C 180,E1 -13366.269,E2 -13366.269} C_VEL
LIN {X 0,Y 356.962,Z 255.824,A -85,B 0,C 180,E1 -13370.161,E2 -13370.161} C_VEL
LIN {X 0,Y 357.616,Z 260.85,A -85,B 0,C 180,E1 -13373.143,E2 -13373.143} C_VEL
LIN {X 0,Y 357.235,Z 265.568,A -85,B 0,C 180,E1 -13375.718,E2 -13375.718} C_VEL
LIN {X 0,Y 356.363,Z 272.159,A -85,B 0,C 180,E1 -13379.154,E2 -13379.154} C_VEL
LIN {X 0,Y 355.574,Z 279.668,A -85,B 0,C 180,E1 -13382.963,E2 -13382.963} C_VEL
LIN {X 0,Y 354.827,Z 287.191,A -85,B 0,C 180,E1 -13386.665,E2 -13386.665} C_VEL
LIN {X 0,Y 354.455,Z 292.455,A -85,B 0,C 180,E1 -13389.234,E2 -13389.234} C_VEL
LIN {X 0,Y 357.179,Z 306.207,A -85,B 0,C 180,E1 -13389.899,E2 -13389.899} C_VEL
LIN {X 0,Y 358.909,Z 318.993,A -85,B 0,C 180,E1 -13390.71,E2 -13390.71} C_VEL
